				Out_uiAktSchritt := In_uiSchritt_09;
			ELSIF	(InOut_uiStatus_10 <> 0)
					AND (InOut_uiStatus_10 <> 4) THEN
				Out_uiAktSchritt := In_uiSchritt_10;				
			ELSIF	(InOut_uiStatus_11 <> 0)						(* 2014-07 gt: RDK90 *)
					AND (InOut_uiStatus_11 <> 4) THEN				(* 2014-07 gt: RDK90 *)
				Out_uiAktSchritt := In_uiSchritt_11;				(* 2014-07 gt: RDK90 *)
			ELSIF	(InOut_uiStatus_12 <> 0)						(* 2014-07 gt: RDK90 *)
					AND (InOut_uiStatus_12 <> 4) THEN				(* 2014-07 gt: RDK90 *)
				Out_uiAktSchritt := In_uiSchritt_12;				(* 2014-07 gt: RDK90 *)
			ELSIF	(InOut_uiStatus_13 <> 0)						(* 2014-07 gt: RDK90 *)
					AND (InOut_uiStatus_13 <> 4) THEN				(* 2014-07 gt: RDK90 *)
				Out_uiAktSchritt := In_uiSchritt_13;				(* 2014-07 gt: RDK90 *)
			ELSIF	(InOut_uiStatus_14 <> 0)						(* 2014-07 gt: RDK90 *)
					AND (InOut_uiStatus_14 <> 4) THEN				(* 2014-07 gt: RDK90 *)
				Out_uiAktSchritt := In_uiSchritt_14;				(* 2014-07 gt: RDK90 *)
			ELSIF	(InOut_uiStatus_15 <> 0)						(* 2014-07 gt: RDK90 *)
					AND (InOut_uiStatus_15 <> 4) THEN				(* 2014-07 gt: RDK90 *)
				Out_uiAktSchritt := In_uiSchritt_15;				(* 2014-07 gt: RDK90 *)
			ELSIF	(InOut_uiStatus_16 <> 0)						(* 2014-07 gt: RDK90 *)
					AND (InOut_uiStatus_16 <> 4) THEN				(* 2014-07 gt: RDK90 *)
				Out_uiAktSchritt := In_uiSchritt_16;				(* 2014-07 gt: RDK90 *)
			ELSIF	(InOut_uiStatus_17 <> 0)						(* 2014-07 gt: RDK90 *)
					AND (InOut_uiStatus_17 <> 4) THEN				(* 2014-07 gt: RDK90 *)
				Out_uiAktSchritt := In_uiSchritt_17;				(* 2014-07 gt: RDK90 *)
			ELSIF	(InOut_uiStatus_18 <> 0)						(* 2016-09 gt: *)
					AND (InOut_uiStatus_18 <> 4) THEN				(* 2016-09 gt: *)
				Out_uiAktSchritt := In_uiSchritt_18;				(* 2016-09 gt: *)
			ELSIF	(uiStatus_19_in_out <> 0)						(* 2016-09 gt: *)
					AND (uiStatus_19_in_out <> 4) THEN				(* 2016-09 gt: *)
				Out_uiAktSchritt := In_uiSchritt_19;				(* 2016-09 gt: *)
			ELSIF	(uiStatus_20_in_out <> 0)						(* 2016-09 gt: *)
					AND (uiStatus_20_in_out <> 4) THEN				(* 2016-09 gt: *)
				Out_uiAktSchritt := In_uiSchritt_20;				(* 2016-09 gt: *)
			ELSIF	(uiStatus_21_in_out <> 0)						(* 2016-09 gt: *)
					AND (uiStatus_21_in_out <> 4) THEN				(* 2016-09 gt: *)
				Out_uiAktSchritt := In_uiSchritt_21;				(* 2016-09 gt: *)
			END_IF
	ELSE Out_uiAktSchritt := 0;								
	END_IF
	(********************************************************************************************************************************************************)
	(* Transition / Weiterschaltung, wenn Einzelschritte beendet oder nicht relevant ************************************************************************)
	IF	TRUE
		AND	(	InOut_uiStatus_01 = 0
				OR InOut_uiStatus_01 = 3
				OR InOut_uiStatus_01 = 4								(* input/output: Status "1" *)
			)
		AND	(	InOut_uiStatus_02 = 0
				OR InOut_uiStatus_02 = 3
				OR InOut_uiStatus_02 = 4								(* input/output: Status "1" *)
			)		
		AND	(	InOut_uiStatus_03 = 0
				OR InOut_uiStatus_03 = 3
				OR InOut_uiStatus_03 = 4								(* input/output: Status "1" *)
			)
		AND	(	InOut_uiStatus_04 = 0
				OR InOut_uiStatus_04 = 3
				OR InOut_uiStatus_04 = 4								(* input/output: Status "1" *)
			)		
		AND	(	InOut_uiStatus_05 = 0
				OR InOut_uiStatus_05 = 3
				OR InOut_uiStatus_05 = 4								(* input/output: Status "1" *)
			)		
		AND	(	InOut_uiStatus_06 = 0
				OR InOut_uiStatus_06 = 3
				OR InOut_uiStatus_06 = 4								(* input/output: Status "1" *)
			)		
		AND	(	InOut_uiStatus_07 = 0
				OR InOut_uiStatus_07 = 3
				OR InOut_uiStatus_07 = 4								(* input/output: Status "1" *)
			)		
		AND	(	uiStatus_08_in_out = 0
				OR uiStatus_08_in_out = 3
				OR uiStatus_08_in_out = 4								(* input/output: Status "1" *)
			)		
		AND	(	InOut_uiStatus_09 = 0
				OR InOut_uiStatus_09 = 3
				OR InOut_uiStatus_09 = 4								(* input/output: Status "1" *)
			)		
		AND	(	InOut_uiStatus_10 = 0
				OR InOut_uiStatus_10 = 3
				OR InOut_uiStatus_10 = 4								(* input/output: Status "1" *)
			)
		AND	(	InOut_uiStatus_11 = 0																		(* 2014-07 gt: RDK90 *)
				OR InOut_uiStatus_11 = 3																	(* 2014-07 gt: RDK90 *)
				OR InOut_uiStatus_11 = 4								(* input/output: Status "1" *)		(* 2014-07 gt: RDK90 *)
			)																
		AND	(	InOut_uiStatus_12 = 0																		(* 2014-07 gt: RDK90 *)
				OR InOut_uiStatus_12 = 3																	(* 2014-07 gt: RDK90 *)
				OR InOut_uiStatus_12 = 4								(* input/output: Status "1" *)		(* 2014-07 gt: RDK90 *)
			)	
		AND	(	InOut_uiStatus_13 = 0																		(* 2014-07 gt: RDK90 *)
				OR InOut_uiStatus_13 = 3																	(* 2014-07 gt: RDK90 *)
				OR InOut_uiStatus_13 = 4								(* input/output: Status "1" *)		(* 2014-07 gt: RDK90 *)
			)	
		AND	(	InOut_uiStatus_14 = 0																		(* 2014-07 gt: RDK90 *)
				OR InOut_uiStatus_14 = 3																	(* 2014-07 gt: RDK90 *)
				OR InOut_uiStatus_14 = 4								(* input/output: Status "1" *)		(* 2014-07 gt: RDK90 *)
			)	
		AND	(	InOut_uiStatus_15 = 0																		(* 2014-07 gt: RDK90 *)
				OR InOut_uiStatus_15 = 3																	(* 2014-07 gt: RDK90 *)
				OR InOut_uiStatus_15 = 4								(* input/output: Status "1" *)		(* 2014-07 gt: RDK90 *)
			)
		AND	(	InOut_uiStatus_16 = 0																		(* 2014-07 gt: RDK90 *)
				OR InOut_uiStatus_16 = 3																	(* 2014-07 gt: RDK90 *)
				OR InOut_uiStatus_16 = 4								(* input/output: Status "1" *)		(* 2014-07 gt: RDK90 *)
			)
		AND	(	InOut_uiStatus_17 = 0																		(* 2014-07 gt: RDK90 *)
				OR InOut_uiStatus_17 = 3																	(* 2014-07 gt: RDK90 *)
				OR InOut_uiStatus_17 = 4								(* input/output: Status "1" *)		(* 2014-07 gt: RDK90 *)
			)
		AND	(	InOut_uiStatus_18 = 0																		(* 2016-09 gt: *)
				OR InOut_uiStatus_18 = 3																	(* 2016-09 gt: *)
				OR InOut_uiStatus_18 = 4								(* input/output: Status "1" *)		(* 2016-09 gt: *)
			)
		AND	(	uiStatus_19_in_out = 0																		(* 2016-09 gt: *)
				OR uiStatus_19_in_out = 3																	(* 2016-09 gt: *)
				OR uiStatus_19_in_out = 4								(* input/output: Status "1" *)		(* 2016-09 gt: *)
			)
		AND	(	uiStatus_20_in_out = 0																		(* 2016-09 gt: *)
				OR uiStatus_20_in_out = 3																	(* 2016-09 gt: *)
				OR uiStatus_20_in_out = 4								(* input/output: Status "1" *)		(* 2016-09 gt: *)
			)
		AND	(	uiStatus_21_in_out = 0																		(* 2016-09 gt: *)
				OR uiStatus_21_in_out = 3																	(* 2016-09 gt: *)
				OR uiStatus_21_in_out = 4								(* input/output: Status "1" *)		(* 2016-09 gt: *)
			) THEN		
		Out_bTransistion := TRUE;		
		Out_uiAktSchritt := In_uiSchrittTransition;					(* Schrittnummer für die Transition nach Blockquittierung, wenn also der Block abgearbeitet ist *)
	ELSE
		Out_bTransistion := FALSE;
	END_IF
ELSE
	In_uiSchritt_01					:= 0;								(* input: Schrittnummer "1" *)
	In_uiSchritt_02					:= 0;								(* input: Schrittnummer "2" *)
	In_uiSchritt_03					:= 0;								(* input: Schrittnummer "3" *)
	In_uiSchritt_04					:= 0;								(* input: Schrittnummer "4" *)
	In_uiSchritt_05					:= 0;								(* input: Schrittnummer "5" *)
	In_uiSchritt_06					:= 0;								(* input: Schrittnummer "6" *)	
	In_uiSchritt_07					:= 0;								(* input: Schrittnummer "7" *)
	In_uiSchritt_08					:= 0;								(* input: Schrittnummer "8" *)
	In_uiSchritt_09					:= 0;								(* input: Schrittnummer "9" *)
	In_uiSchritt_10					:= 0;								(* input: Schrittnummer "10" *)	
	In_uiSchritt_11					:= 0;								(* input: Schrittnummer "11" *)			(* 2014-07 gt: RDK90 *)
	In_uiSchritt_12					:= 0;								(* input: Schrittnummer "12" *)			(* 2014-07 gt: RDK90 *)
	In_uiSchritt_13					:= 0;								(* input: Schrittnummer "13" *)			(* 2014-07 gt: RDK90 *)
	In_uiSchritt_14					:= 0;								(* input: Schrittnummer "14" *)			(* 2014-07 gt: RDK90 *)
	In_uiSchritt_15					:= 0;								(* input: Schrittnummer "15" *)			(* 2014-07 gt: RDK90 *)
	In_uiSchritt_16					:= 0;								(* input: Schrittnummer "16" *)			(* 2014-07 gt: RDK90 *)
	In_uiSchritt_17					:= 0;								(* input: Schrittnummer "17" *)			(* 2014-07 gt: RDK90 *)
	In_uiSchritt_18					:= 0;								(* input: Schrittnummer "18" *)			(* 2016-09 gt: *)
	In_uiSchritt_19					:= 0;								(* input: Schrittnummer "19" *)			(* 2016-09 gt: *)
	In_uiSchritt_20					:= 0;								(* input: Schrittnummer "20" *)			(* 2016-09 gt: *)
	In_uiSchritt_21					:= 0;								(* input: Schrittnummer "21" *)			(* 2016-09 gt: *)	

	InOut_bQuit_01					:= FALSE;							(* input/output: Quittierung "1" *)
	InOut_uiStatus_01				:= 0;								(* input/output: Status "1" *)
	InOut_bQuit_02					:= FALSE;							(* input/output: Quittierung "2" *)	
	InOut_uiStatus_02				:= 0;								(* input/output: Status "2" *)
	InOut_bQuit_03					:= FALSE;							(* input/output: Quittierung "3" *)
	InOut_uiStatus_03				:= 0;								(* input/output: Status "3" *)
	InOut_bQuit_04					:= FALSE;							(* input/output: Quittierung "4" *)	
	InOut_uiStatus_04				:= 0;								(* input/output: Status "4" *)
	InOut_bQuit_05					:= FALSE;							(* input/output: Quittierung "5" *)
	InOut_uiStatus_05				:= 0;								(* input/output: Status "5" *)
	InOut_bQuit_06					:= FALSE;							(* input/output: Quittierung "6" *)	
	InOut_uiStatus_06				:= 0;								(* input/output: Status "6" *)
	InOut_bQuit_07					:= FALSE;							(* input/output: Quittierung "7" *)
	InOut_uiStatus_07				:= 0;								(* input/output: Status "7" *)
	InOut_bQuit_08					:= FALSE;							(* input/output: Quittierung "8" *)	
	uiStatus_08_in_out				:= 0;								(* input/output: Status "8" *)
	InOut_bQuit_09					:= FALSE;							(* input/output: Quittierung "9" *)
	InOut_uiStatus_09				:= 0;								(* input/output: Status "9" *)
	InOut_bQuit_10					:= FALSE;							(* input/output: Quittierung "10" *)		
	InOut_uiStatus_10				:= 0;								(* input/output: Status "10" *)
	InOut_bQuit_11					:= FALSE;							(* input/output: Quittierung "11" *)	(* 2014-07 gt: RDK90 *)		
	InOut_uiStatus_11				:= 0;								(* input/output: Status "11" *)			(* 2014-07 gt: RDK90 *)
	InOut_bQuit_12					:= FALSE;							(* input/output: Quittierung "12" *)	(* 2014-07 gt: RDK90 *)	
	InOut_uiStatus_12				:= 0;								(* input/output: Status "12" *)			(* 2014-07 gt: RDK90 *)
	InOut_bQuit_13					:= FALSE;							(* input/output: Quittierung "13" *)	(* 2014-07 gt: RDK90 *)	
	InOut_uiStatus_13				:= 0;								(* input/output: Status "13" *)			(* 2014-07 gt: RDK90 *)
	InOut_bQuit_14					:= FALSE;							(* input/output: Quittierung "14" *)	(* 2014-07 gt: RDK90 *)	
	InOut_uiStatus_14				:= 0;								(* input/output: Status "14" *)			(* 2014-07 gt: RDK90 *)
	InOut_bQuit_15					:= FALSE;							(* input/output: Quittierung "15" *)	(* 2014-07 gt: RDK90 *)	
	InOut_uiStatus_15				:= 0;								(* input/output: Status "15" *)			(* 2014-07 gt: RDK90 *)
	InOut_bQuit_16					:= FALSE;							(* input/output: Quittierung "16" *)	(* 2014-07 gt: RDK90 *)	
	InOut_uiStatus_16				:= 0;								(* input/output: Status "16" *)			(* 2014-07 gt: RDK90 *)	
	InOut_bQuit_17					:= FALSE;							(* input/output: Quittierung "17" *)	(* 2014-07 gt: RDK90 *)	
	InOut_uiStatus_17				:= 0;								(* input/output: Status "17" *)			(* 2014-07 gt: RDK90 *)
	InOut_bQuit_18					:= FALSE;							(* input/output: Quittierung "18" *)	(* 2016-09 gt: *)	
	InOut_uiStatus_18				:= 0;								(* input/output: Status "18" *)			(* 2016-09 gt: *)
	bQuit_19_in_out					:= FALSE;							(* input/output: Quittierung "19" *)	(* 2016-09 gt: *)	
	uiStatus_19_in_out				:= 0;								(* input/output: Status "19" *)			(* 2016-09 gt: *)
	bQuit_20_in_out					:= FALSE;							(* input/output: Quittierung "20" *)	(* 2016-09 gt: *)	
	uiStatus_20_in_out				:= 0;								(* input/output: Status "20" *)			(* 2016-09 gt: *)
	bQuit_21_in_out					:= FALSE;							(* input/output: Quittierung "21" *)	(* 2016-09 gt: *)	
	uiStatus_21_in_out				:= 0;								(* input/output: Status "21" *)			(* 2016-09 gt: *)	
	
	Out_uiAktSchritt				:= 0;								(* output: Aktueller Schritt aufgrund der "höchswertigsten" Quittierung  *)
	Out_bTransistion				:= FALSE;							(* output: Transition / Weiterschaltung, wenn Einzelschritte beendet oder nicht relevant *)	
END_IF	
(********************************************************************************************************************************************************)

END_FUNCTION_BLOCK

// GeneralFunctionBlocks/FB_ClockMarker
{attribute 'qualified_only' := ''}
{attribute 'namespace' := 'ILGStdLib.FunctionBlocks'}
FUNCTION_BLOCK FB_ClockMarker
VAR_OUTPUT
	/// Ausgangsvariable, die in der anparametrierten rRDM_Taktzeit_gb taktet 
	Out_bClock: BOOL;
	/// Ausgangsvariable, die in der anparametrierten rRDM_Taktzeit_gb einen Impuls abgibt 
	Out_bPulse: BOOL;
END_VAR
VAR
	/// Funktionsbaustein "Einschaltverzoegerung" fuer den Taktmerker 
	fbTonClock1: TON;
	/// Funktionsbaustein "Einschaltverzoegerung" fuer den Taktmerker 
	fbTonClock2: TON;
	/// Funktionsbaustein positive Flanke für Taktmerker 
	rtrig_Clock: R_TRIG;
END_VAR
VAR_INPUT
	/// Ansteuersignal fuer den Start des Funktionsbausteins / das Erzeugen das Taktimpulses 
	In_bEnable: BOOL;
	/// Anzuparametrierende Zeit, fuer die rRDM_Taktzeit_gb 
	In_tCycleTime: TIME;
END_VAR

(* #################################################################################################################### *)
(* ##   iLLiG_FB_Taktmerker	    																				 	 ## *)
(* ##																												 ## *)
(* ##	Dieser Funktionsbaustein erzeugt ein taktendes Ausgangssignal, in Abhaengigkeit der anparametrierten	     ## *)
(* ##	Zeitdauer.																									 ## *)
(* ##																												 ## *)
(* ##   Versions-History:																							 ## *)
(* ##   06. Dezember 2011		Version 1.0		-	erste Version.													 ## *)
(* ##																												 ## *)
(* ##																												 ## *)
(* #################################################################################################################### *)


(* -------------------------------------------------------------------------------------------------------------------- *)
(* -- Erzeugen des Taktsignals ---------------------------------------------------------------------------------------- *)	
(* -------------------------------------------------------------------------------------------------------------------- *)

IF In_bEnable THEN

	fbTonClock1(IN:= (NOT Out_bClock), PT:= In_tCycleTime, Q=> , ET=> );					(* Aufruf der Einschaltverzoegerung 1 *)
		
	fbTonClock2(IN:= (Out_bClock), PT:= In_tCycleTime, Q=> , ET=> );						(* Aufruf der Einschaltverzoegerung 2 *)
	
	IF fbTonClock1.Q THEN
		Out_bClock := TRUE;																(* Ausgang setzen *)
	ELSIF fbTonClock2.Q THEN
		Out_bClock := FALSE;																(* Ausgang zurueck setzen *)
	END_IF
	
	(* Impuls von Takt bilden *)
	rtrig_Clock(CLK:= Out_bClock);
	Out_bPulse := rtrig_Clock.Q;
	
ELSE
	Out_bClock		:= FALSE;															(* Ausgang abloeschen *)
	fbTonClock1(IN:= FALSE, PT:= In_tCycleTime, Q=> , ET=> );							(* Funktionsbaustein zurueck setzen *)
	fbTonClock2(IN:= FALSE, PT:= In_tCycleTime, Q=> , ET=> );							(* Funktionsbaustein zurueck setzen *)
END_IF

END_FUNCTION_BLOCK

// GeneralFunctionBlocks/FB_Convert8BitTo5BitParameter
{attribute 'qualified_only' := ''}
{attribute 'namespace' := 'ILGStdLib.FunctionBlocks'}
FUNCTION_BLOCK FB_Convert8BitTo5BitParameter
VAR_OUTPUT
	Out_dwOutput: DWORD;
	Out_bDone: BOOL;
	Out_bError: BOOL;
	Out_bActive: BOOL;
END_VAR
VAR
	udiTemp: UDINT;
	udiInput: UDINT;
	iStep: INT;
END_VAR
VAR_INPUT
	In_diInput: DINT;
	In_udiMask: UDINT;
	In_bEnable: BOOL;
	In_bStart: BOOL;
END_VAR

(* #################################################################################################################### *)
(* ##   iLLiG_FB_Bremspruefung    																				 	 ## *)
(* ##																											     ## *)
(* ##   erstellt von:																								 ## *)
(* ##   Markus Pfisterer, EE																						 ## *)
(* ##																											     ## *)
(* ##   Versions-History:																							 ## *)
(* ##   12.Oktober 2018		Version 1.0		-	Erste Version, nach Bereinigung der Fehler							 ## *)
(* #################################################################################################################### *)

(*
Funktionsbeschreibung:
Der Baustein konvertiert den Parameter S-0-0390 in ein bekanntes fünfstelliges Format.
*)


(* ####################################################################################################################################### *)
IF In_bEnable THEN
	(* #################################################### *)
	(* Start der Schritkette *)
	IF In_bStart AND NOT Out_bActive THEN
		iStep := 10;
	END_IF

	(* #################################################### *)
	(* Statusmeldung bilden *)
	IF iStep > 0 THEN
		Out_bActive := TRUE;
	ELSE
		Out_bActive := FALSE;
	END_IF


	(* #################################################### *)
	(* Schrittkette zur Konvertierung *)
	CASE iStep OF
	
		(* Initialisierung des Bausteins *)
		10:
			Out_bDone  := FALSE;
			Out_bError := FALSE;
			iStep 	 := 20;
			
		(* Konvertierung *)
		20:
			udiInput := DINT_TO_UDINT(In_diInput AND 16#000FFFFF);
			
			IF udiInput > 16#000F0000 THEN					// Error
				udiTemp := udiInput AND 16#00FF0000;			// Check if Error comes from IndraDrive 
				IF udiTemp = 16#F0000 THEN
					udiInput := udiInput AND In_udiMask;
					Out_dwOutput := udiInput + 16#000F0000;
					Out_bDone    := TRUE;
				ELSE
					Out_dwOutput := DINT_TO_DWORD(16#0);
					Out_bError    := TRUE;	
				END_IF	
				
			ELSIF udiInput > 16#000E0000 THEN				// Warning
				udiTemp := udiInput AND  16#00FF0000;			// Check if Error comes from IndraDrive 
				IF udiTemp = 16#E0000 THEN
					udiInput := udiInput AND In_udiMask;
					Out_dwOutput := udiInput + 16#000E0000;
					Out_bDone    := TRUE;
				ELSE
					Out_dwOutput := DINT_TO_DWORD(16#0);	
					Out_bError    := TRUE;	
				END_IF	
			ELSIF udiInput > 16#000C0000 THEN				// Diagnosis
				udiTemp := udiInput AND  16#00FF0000;			// Check if Error comes from IndraDrive 
				IF udiTemp = 16#C0000 THEN
					udiInput := udiInput AND In_udiMask;
					Out_dwOutput := udiInput + 16#000C0000;
					Out_bDone    := TRUE;
				ELSE
					Out_dwOutput := DINT_TO_DWORD(16#0);
					Out_bError    := TRUE;		
				END_IF
			ELSIF udiInput > 16#000A0000 THEN				// Status
				udiTemp := udiInput AND  16#00FF0000;			// Check if Error comes from IndraDrive 
				IF udiTemp = 16#A0000 THEN
					udiInput := udiInput AND In_udiMask;
					Out_dwOutput := udiInput + 16#000A0000;
					Out_bDone    := TRUE;
				ELSE
					Out_dwOutput := DINT_TO_DWORD(16#0);
					Out_bError    := TRUE;		
				END_IF
				
			ELSE
				Out_bError := TRUE;	
			END_IF
	
			Out_bActive := FALSE;
			iStep 	  := 0;
	END_CASE
END_IF

END_FUNCTION_BLOCK

// GeneralFunctionBlocks/FB_IlligOperatingModes
{attribute 'qualified_only' := ''}
{attribute 'namespace' := 'ILGStdLib.FunctionBlocks'}
FUNCTION_BLOCK FB_IlligOperatingModes
VAR_OUTPUT
	/// Dummyvariable, da bei erster Variable keine Quick Info möglich 
	OUT_bDummy: BOOL;
	/// Betriebsart: "Referenzieren" (M12.7) 
	OUT_bBetriebsart_Ctrl_REFERENZIEREN: BOOL;
	/// Betriebsart: Vorwahl "Referenzieren" (M12.6) 
	OUT_bBetriebsart_Vorwahl_REFERENZIEREN: BOOL;
	/// Betriebsart: "Hand" (M13.0)
	OUT_bBetriebsart_Ctrl_HAND: BOOL;
	/// Betriebsart: "Ruesten" (M12.0) 
	OUT_bBetriebsart_Ctrl_RUESTEN: BOOL;
	/// Betriebsart: "Einruesten" (M12.1) 
	OUT_bBetriebsart_Ctrl_EINRUESTEN: BOOL;
	/// Betriebsart: "Ausruesten" (M12.2) 
	OUT_bBetriebsart_Ctrl_AUSRUESTEN: BOOL;
	/// Betriebsart: "VorwahlAuto" (M14.7)
	OUT_bBetriebsart_Ctrl_VORWAHLAUTO: BOOL;
	/// Betriebsart: "Automatik" oder "Startautomatik" ("M14.5" oder "M18.3")
	OUT_bBetriebsart_Ctrl_AUTOLAEUFT: BOOL;
	/// Betriebsart: "Automatik" (M14.0)
	OUT_bBetriebsart_Ctrl_AUTOMATIK: BOOL;
	/// Betriebsart: "Grundstellungsfahrt" (M14.4)
	OUT_bBetriebsart_Ctrl_GRUNDSTELLUNGSFAHRT: BOOL;
	/// Betriebsart: "Automatik Laeuft" und "Startautomatik" beendet (M14.5) 
	OUT_bBetriebsart_Ctrl_AUTOLAEUFT_STARTAUTO_fertig: BOOL;
	/// Betriebsart: "Schluesselschalter" (M11.7) 
	OUT_bBetriebsart_Ctrl_SCHLUESSELSCHALTER: BOOL;
	/// Betriebsart: Impuls Drucktaster "Start" (M11.0) 
	OUT_bImp_DT_Automatik_Start: BOOL;
	/// Betriebsart: Impuls "Automatik EIN" (M16.0) 
	OUT_bImp_Betriebsart_Ctrl_AUTOMATIK_EIN: BOOL;
	/// Betriebsart: Impuls "Automatik AUS" (M16.2) 
	OUT_bImp_Betriebsart_Ctrl_AUTOMATIK_AUS: BOOL;
	/// Betriebsart: Impuls "Automatik Laeuft" und "Startautomatik" beendet (M16.4) 
	OUT_bImp_Betriebsart_Ctrl_AUTOLAEUFT_STARTAUTO_fertig: BOOL;
	/// Betriebsart: "Automatik Aus" (nicht M14.0 und nicht M14.5) verzögert 1 Sek. 
	OUT_bBetriebsart_Automatik_Aus_Verz: BOOL;
	/// Betriebsart: Freigabe Hand (M13.1) 
	OUT_bFreig_Betriebsart_Hand: BOOL;
	/// Anforderung Stop in Grundstellung gespeichert 
	OUT_bAnf_StopGrdst_gesp: BOOL;
	/// Anzeige Betriebsart: 0= Hand, 1= Rüsten, 2= Einrüsten, 4= Ausrüsten, 8= Vorwahl Automatik, 16= Vorwahl Referenzieren 
	OUT_byAnzeige_Betriebsart: BYTE;
END_VAR
VAR
	/// Dummyvariable, da bei erster Variable keine Quick Info möglich 
	bDummy: BOOL;
	/// Bedienfeld Anwahl "Vorwahl Automatik" 
	bBBF_Anw_Betriebsart_Automatik: BOOL;
	/// Bedienfeld Anwahl Betriebsart Hand 
	bBBF_Anw_Betriebsart_Hand: BOOL;
	/// Impuls Grundstellungsfahrt beendet (M17.2) 
	bImpuls_GrdstFahrt_Beendet: BOOL;
	/// Freigabe Grundstellungsfahrt 
	bFreig_Grundstellungsfahrt: BOOL;
	/// Start Grundstellungsfahrt exter gespeichert 
	bStart_Grundstellungsfahrt_extern_gesp: BOOL;
	/// Anforderung Stop in Grundstellung gespeichert 
	bAnf_StopGrdst_gesp: BOOL;
	/// Dummyvariable, da bei erster Variable keine Quick Info möglich 
	rtrigDummy: R_TRIG;
	/// Positive Flanke Bedienfeld Anwahl Schlüsselschalter ( M19.6) 
	rtrigBetriebsart_Ctrl_Schluesselschalter: R_TRIG;
	/// Negative Flanke Bedienfeld Anwahl Schlüsselschalter ( M19.2) 
	ftrigBetriebsart_Ctrl_Schluesselschalter: F_TRIG;
	/// Positive Flanke Drucktaster Automatik Start (M11.0)
	rtrigDT_Automatik_Start: R_TRIG;
	/// Positive Flanke Drucktaster Automatik Stop (M11.2)
	rtrigDT_Automatik_Stop: R_TRIG;
	/// Positive Flanke Bedienfeld Anwahl Betriebsart Ruesten ( M27.0) 
	rtrigBBF_Anw_Betriebsart_Ruesten: R_TRIG;
	/// Positive Flanke Bedienfeld Anwahl Betriebsart Einruesten ( M27.1) 
	rtrigBBF_Anw_Betriebsart_Einruesten: R_TRIG;
	/// Positive Flanke Bedienfeld Anwahl Betriebsart Ausruesten ( M27.2) 
	rtrigBBF_Anw_Betriebsart_Ausruesten: R_TRIG;
	/// Positive Flanke Bedienfeld Anwahl Betriebsart Referenzieren ( M27.3) 
	rtrigBBF_Anw_Betriebsart_Referenzieren: R_TRIG;
	/// Hilfsmerker für Impuls Grundstellungsfahrt beendet 
	rtrigHM_Impuls_Grundstellungsfahrt_beendet: R_TRIG;
	/// Hilfsmerker Positive Flanke "Automatik EIN" 
	rtrigHM_Automatik_EIN: R_TRIG;
	/// Hilfsmerker Positive Flanke "Automatik AUS" 
	rtrigHM_Automatik_AUS: R_TRIG;
	/// Hilfsmerker Positive Flanke "Automatik läuft" 
	rtrigHM_Automatik_laeuft: R_TRIG;
	/// Hilfsmerker "Automatik AUS" verzögert 
	tonHM_Automatik_Aus: TON;
	/// Hilfsmerker Positive Flanke Impuls "Automatik Laeuft" und "Startautomatik" beendet 
	rtrigHM_AUTOLAEUFT_STARTAUTO_fertig: R_TRIG;
END_VAR
VAR_INPUT
	/// Dummyvariable, da bei erster Variable keine Quick Info möglich 
	IN_bDummy: BOOL;
	/// Drucktaster "Betriebsart Start" 
	IN_bDT_Betriebsart_Start: BOOL;
	/// Drucktaster "Betriebsart Stop" 
	IN_bDT_Betriebsart_Stop: BOOL;
	/// Schlüsselschalter 
	IN_bSCHLUESSELSCHALTER: BOOL;
	/// Bedienfeld Anwahl Betriebsart Ruesten ( M27.0) 
	IN_bBBF_Anw_Betriebsart_Ruesten: BOOL;
	/// Bedienfeld Anwahl Betriebsart Einruesten ( M27.1) 
	IN_bBBF_Anw_Betriebsart_Einruesten: BOOL;
	/// Bedienfeld Anwahl Betriebsart Ausruesten ( M27.2) 
	IN_bBBF_Anw_Betriebsart_Ausruesten: BOOL;
	/// Bedienfeld Anwahl Betriebsart Referenzieren ( M27.3) 
	IN_bBBF_Anw_Betriebsart_Referenzieren: BOOL;
	/// Linie in Grundstellung (RDM & Stapelung (M14.6) 
	IN_bLinie_In_Grundstellung: BOOL;
	/// Anforderung Vorwahl Automatik extern. Z.B. von Bremsprüfung 
	IN_bAnf_Vorwahl_Automatik_extern: BOOL;
	/// Schrittkette Werkzeugeinbau aktiv (M518.4) 
	IN_bSKWerkzeugeinbau_aktiv: BOOL;
	/// Schrittkette Werkzeugausbau aktiv (M537.7) 
	IN_bSKWerkzeugausbau_aktiv: BOOL;
	/// Ein- und Ausrüsten zurücksetzen 
	IN_bReset_Ein_Ausruesten_extern: BOOL;
	/// Anforderung Betriebsart Hand von extern z.B. von Bremsprüfung 
	IN_bAnf_Betriebsart_Hand_extern: BOOL;
	/// Reset Betriebsart Hand von extern z.B. von Bremsprüfung 
	IN_bReset_Betriebsart_Hand_extern: BOOL;
	/// Reset Vorwahl Automatik von extern z.B. von Bremsprüfung 
	IN_bReset_Vorwahl_Automatik_extern: BOOL;
	/// Freigabe Vorwahl Automatik 
	IN_bFreig_Vorwahl_Automatik_extern: BOOL;
	/// Stopp in Grundstellung Fehler aktiv 
	IN_bStopInGrundstellung: BOOL;
	/// Sofortstopfehler aktiv 
	IN_bSofortstopp: BOOL;
	/// Abläufe in Vorwahl Automatik aktiv z.B. Räumen 
	IN_bAblaeufe_Vorwahl_Automatik_aktiv: BOOL;
	/// Steuerstrom EIN (M10.0) 
	IN_bSteuerstrom_Ein: BOOL;
	/// Freigabe Grundstellungsfahrt 
	IN_bFreig_Grundstellungsfahrt_extern: BOOL;
	/// Freigabe Grundstellungsfahrt ohne Schlüsselschalter (Bsp. innerhalb des Rüstablaufs 
	IN_bFreig_GrdstFahrt_mit_SCHLUESSELSCHALTER_extern: BOOL;
	/// Grundstellungsfahrt löschen extern
	IN_bGrdstFahrt_loeschen_extern: BOOL;
	/// Anforderung Grundstellungsfahrt von Extern z.B.Bremsprüfung 
	IN_bAnf_Grundstellungsfahrt_Extern: BOOL;
	/// Reset Automatik von Extern z.B. Bremsprüfung, Schmierhub... 
	IN_bReset_Automatik_extern: BOOL;
	/// Freigabe Automatik 
	IN_bFreig_Automatik_extern: BOOL;
	/// Automatikabläufe der Linie nicht aktiv, Automatik läuft kann zurückgenommen werden 
	IN_bAutomatikablaeufe_nicht_Aktiv: BOOL;
	/// Freigabe "Automatik läuft" extern 
	IN_bFreig_Automatik_Laeuft_extern: BOOL;
	/// Freigabe "Automatik Stopp in Grundstellung" extern 
	IN_bFreig_Automatik_Stop_Grdst_extern: BOOL;
	/// Start "Automatik läuft" Extern 
	IN_bStart_Automatik_Laeuft_Extern: BOOL;
	/// Startautomatik läuft 
	IN_bStartautomatik_Laeuft: BOOL;
END_VAR


(*##########################################################################################################################################################################################################*)
(* Drucktaster, Schlüsselschalter, BBF-Anwahlen *)
(*##########################################################################################################################################################################################################*)

(* Positive Flanke Drucktaster "Start" *)
rtrigDT_Automatik_Start(CLK:= IN_bDT_Betriebsart_Start);

(* Positive Flanke Drucktaster "Stop" *)
rtrigDT_Automatik_Stop(CLK:= IN_bDT_Betriebsart_Stop);

(* Schluesselschalter eingeschaltet *)
OUT_bBetriebsart_Ctrl_SCHLUESSELSCHALTER := IN_bSCHLUESSELSCHALTER AND NOT OUT_bBetriebsart_Ctrl_AUTOLAEUFT;

(* Positive Flanke Bedienfeld Anwahl Schluesselschalter *)
rtrigBetriebsart_Ctrl_Schluesselschalter(CLK:= IN_bSCHLUESSELSCHALTER);

(* Negative Flanke Bedienfeld Anwahl Schluesselschalter *)
ftrigBetriebsart_Ctrl_Schluesselschalter(CLK:= IN_bSCHLUESSELSCHALTER);

(* Positive Flanke Bedienfeld Anwahl Betriebsart Ruesten *)
rtrigBBF_Anw_Betriebsart_Ruesten(CLK:= IN_bBBF_Anw_Betriebsart_Ruesten);

(* Positive Flanke Bedienfeld Anwahl Betriebsart Einruesten *)
rtrigBBF_Anw_Betriebsart_Einruesten(CLK:= IN_bBBF_Anw_Betriebsart_Einruesten);

(* Positive Flanke Bedienfeld Anwahl Betriebsart Ausruesten *)
rtrigBBF_Anw_Betriebsart_Ausruesten(CLK:= IN_bBBF_Anw_Betriebsart_Ausruesten);

(* Positive Flanke Bedienfeld Anwahl Betriebsart Referenzieren *)
rtrigBBF_Anw_Betriebsart_Referenzieren(CLK:= IN_bBBF_Anw_Betriebsart_Referenzieren);

(* Bedienfeld Anwahl Betriebsart Automatik *)
bBBF_Anw_Betriebsart_Automatik := IN_bLinie_In_Grundstellung AND	bImpuls_GrdstFahrt_Beendet AND IN_bFreig_Vorwahl_Automatik_extern;

(* Bedienfeld Anwahl Betriebsart Hand *)
bBBF_Anw_Betriebsart_Hand := NOT OUT_bBetriebsart_Ctrl_AUTOMATIK AND NOT OUT_bBetriebsart_Ctrl_GRUNDSTELLUNGSFAHRT AND NOT 
																OUT_bBetriebsart_Ctrl_AUTOLAEUFT AND NOT OUT_bBetriebsart_Ctrl_VORWAHLAUTO AND NOT
																OUT_bBetriebsart_Ctrl_SCHLUESSELSCHALTER AND NOT bBBF_Anw_Betriebsart_Automatik AND NOT
																IN_bAnf_Vorwahl_Automatik_extern;

(* Automatik Stopp speichern, um an einer definierten Stelle Stopp in Grundstellung einzuleiten *)
IF ((IN_bStopInGrundstellung OR IN_bReset_Automatik_extern OR rtrigDT_Automatik_Stop.Q) AND NOT IN_bFreig_Automatik_Stop_Grdst_extern) THEN
	bAnf_StopGrdst_gesp := TRUE;
END_IF
(* Sobald die Automatik aus ist, speicher wieder rücksetzen *)
IF NOT OUT_bBetriebsart_Ctrl_AUTOMATIK THEN
	bAnf_StopGrdst_gesp := FALSE;
END_IF																
(*##########################################################################################################################################################################################################*)
(* Betriebsarten *)
(*##########################################################################################################################################################################################################*)
(* ********************************************************************************************************************** *)
(* Ruesten *)
(* ********************************************************************************************************************** *)
(* Betriebsart: "Ruesten" *)
IF ((NOT OUT_bBetriebsart_Ctrl_SCHLUESSELSCHALTER) OR rtrigBBF_Anw_Betriebsart_Einruesten.Q OR rtrigBBF_Anw_Betriebsart_Ausruesten.Q OR
	rtrigBBF_Anw_Betriebsart_Referenzieren.Q) THEN

	OUT_bBetriebsart_Ctrl_RUESTEN:= FALSE;

ELSIF ((rtrigBBF_Anw_Betriebsart_Ruesten.Q AND NOT IN_bSKWerkzeugeinbau_aktiv AND NOT IN_bSKWerkzeugausbau_aktiv) OR
		rtrigBetriebsart_Ctrl_Schluesselschalter.Q OR (rtrigDT_Automatik_Stop.Q AND (OUT_bBetriebsart_Vorwahl_REFERENZIEREN OR
		OUT_bBetriebsart_Ctrl_REFERENZIEREN))) THEN 
		
	OUT_bBetriebsart_Ctrl_RUESTEN:= TRUE;
END_IF
(* ---------------------------------------------------------------------------------------------------------------------- *)
(* Betriebsart: "Einruesten" *)
IF ((NOT OUT_bBetriebsart_Ctrl_SCHLUESSELSCHALTER) OR ((rtrigBBF_Anw_Betriebsart_Ruesten.Q OR rtrigBBF_Anw_Betriebsart_Ausruesten.Q OR 
	rtrigBBF_Anw_Betriebsart_Referenzieren.Q) AND NOT IN_bSKWerkzeugeinbau_aktiv) OR IN_bReset_Ein_Ausruesten_extern) THEN

	OUT_bBetriebsart_Ctrl_EINRUESTEN:= FALSE;

ELSIF (rtrigBBF_Anw_Betriebsart_Einruesten.Q) THEN 

	OUT_bBetriebsart_Ctrl_EINRUESTEN:= TRUE;

END_IF
(* ---------------------------------------------------------------------------------------------------------------------- *)
(* Betriebsart: "Ausruesten" *)
IF ((NOT OUT_bBetriebsart_Ctrl_SCHLUESSELSCHALTER) OR ((rtrigBBF_Anw_Betriebsart_Ruesten.Q OR rtrigBBF_Anw_Betriebsart_Einruesten.Q OR 
	rtrigBBF_Anw_Betriebsart_Referenzieren.Q) AND NOT IN_bSKWerkzeugausbau_aktiv) OR IN_bReset_Ein_Ausruesten_extern) THEN

	OUT_bBetriebsart_Ctrl_AUSRUESTEN:= FALSE;

ELSIF (rtrigBBF_Anw_Betriebsart_Ausruesten.Q) THEN 

	OUT_bBetriebsart_Ctrl_AUSRUESTEN:= TRUE;

END_IF
(* ********************************************************************************************************************** *)
(* Referenzieren *)
(* ********************************************************************************************************************** *)
(* Betriebsart: "Vorwahl Referenzieren" *)
IF ((NOT OUT_bBetriebsart_Ctrl_SCHLUESSELSCHALTER) OR rtrigBBF_Anw_Betriebsart_Ruesten.Q OR	rtrigBBF_Anw_Betriebsart_Einruesten.Q OR 
	rtrigBBF_Anw_Betriebsart_Ausruesten.Q OR rtrigDT_Automatik_Stop.Q) THEN
			
	OUT_bBetriebsart_Vorwahl_REFERENZIEREN:= FALSE;

ELSIF ((rtrigBBF_Anw_Betriebsart_Referenzieren.Q) AND NOT IN_bSKWerkzeugeinbau_aktiv AND NOT IN_bSKWerkzeugausbau_aktiv) THEN 

	OUT_bBetriebsart_Vorwahl_REFERENZIEREN:= TRUE;

END_IF
(* ---------------------------------------------------------------------------------------------------------------------- *)
(* Betriebsart: "Referenzieren" *)
IF ((NOT OUT_bBetriebsart_Ctrl_SCHLUESSELSCHALTER) OR NOT OUT_bBetriebsart_Vorwahl_REFERENZIEREN OR rtrigDT_Automatik_Stop.Q) THEN

	OUT_bBetriebsart_Ctrl_REFERENZIEREN:= FALSE;

ELSIF ((rtrigDT_Automatik_Start.Q) AND OUT_bBetriebsart_Vorwahl_REFERENZIEREN) THEN 

	OUT_bBetriebsart_Ctrl_REFERENZIEREN:= TRUE;

END_IF
(* ********************************************************************************************************************** *)
(* Hand *)
(* ********************************************************************************************************************** *)
(* Betriebsart: "Hand" *)
IF ((OUT_bBetriebsart_Ctrl_SCHLUESSELSCHALTER) OR IN_bReset_Betriebsart_Hand_extern OR OUT_bBetriebsart_Ctrl_GRUNDSTELLUNGSFAHRT OR
	bBBF_Anw_Betriebsart_Automatik) THEN
	
	OUT_bBetriebsart_Ctrl_HAND:= FALSE;

ELSIF (IN_bAnf_Betriebsart_Hand_extern OR bBBF_Anw_Betriebsart_Hand OR (ftrigBetriebsart_Ctrl_Schluesselschalter.Q)) THEN

	OUT_bBetriebsart_Ctrl_HAND:= TRUE;

END_IF
(* ********************************************************************************************************************** *)
(* Automatik *)
(* ********************************************************************************************************************** *)
(* Betriebsart: "Vorwahl Automatik" *)
IF (OUT_bBetriebsart_Ctrl_SCHLUESSELSCHALTER OR IN_bAnf_Betriebsart_Hand_extern OR bBBF_Anw_Betriebsart_Hand OR
	((rtrigDT_Automatik_Stop.Q OR (IN_bStopInGrundstellung AND IN_bLinie_In_Grundstellung AND NOT IN_bAblaeufe_Vorwahl_Automatik_aktiv) OR 
	OUT_bBetriebsart_Ctrl_GRUNDSTELLUNGSFAHRT OR 
	(NOT IN_bLinie_In_Grundstellung AND NOT IN_bAblaeufe_Vorwahl_Automatik_aktiv)) AND NOT OUT_bBetriebsart_Ctrl_AUTOMATIK AND
	 NOT OUT_bBetriebsart_Ctrl_AUTOLAEUFT)) THEN
	
	OUT_bBetriebsart_Ctrl_VORWAHLAUTO:= FALSE;

ELSIF ((IN_bAnf_Vorwahl_Automatik_extern OR bBBF_Anw_Betriebsart_Automatik) AND IN_bFreig_Vorwahl_Automatik_extern AND
	NOT IN_bStopInGrundstellung) THEN
	
	OUT_bBetriebsart_Ctrl_VORWAHLAUTO:= TRUE;

END_IF
(* ---------------------------------------------------------------------------------------------------------------------- *)
(* Impuls Grundstellungsfahrt beendet und Maschine in Grundstellung *)
rtrigHM_Impuls_Grundstellungsfahrt_beendet(CLK:=  (NOT (rtrigDT_Automatik_Start.Q) AND NOT OUT_bBetriebsart_Ctrl_GRUNDSTELLUNGSFAHRT));
bImpuls_GrdstFahrt_Beendet := (rtrigHM_Impuls_Grundstellungsfahrt_beendet.Q AND IN_bLinie_In_Grundstellung);
(* ---------------------------------------------------------------------------------------------------------------------- *)
(* Freigabe Grundstellungsfahrt *)
bFreig_Grundstellungsfahrt := IN_bFreig_Grundstellungsfahrt_extern AND NOT IN_bLinie_In_Grundstellung;
(* ---------------------------------------------------------------------------------------------------------------------- *)
(* Betriebsart: "Grundstellungsfahrt" *)
IF ((OUT_bBetriebsart_Ctrl_SCHLUESSELSCHALTER AND NOT IN_bFreig_GrdstFahrt_mit_SCHLUESSELSCHALTER_extern) OR IN_bStopInGrundstellung OR IN_bSofortstopp OR OUT_bBetriebsart_Ctrl_AUTOMATIK OR
	rtrigDT_Automatik_Stop.Q OR NOT IN_bSteuerstrom_Ein OR OUT_bBetriebsart_Ctrl_AUTOLAEUFT OR (IN_bGrdstFahrt_loeschen_extern AND bStart_Grundstellungsfahrt_extern_gesp)OR 
	(OUT_bBetriebsart_Ctrl_GRUNDSTELLUNGSFAHRT AND IN_bLinie_In_Grundstellung)) THEN

	OUT_bBetriebsart_Ctrl_GRUNDSTELLUNGSFAHRT:= FALSE;
	bStart_Grundstellungsfahrt_extern_gesp := FALSE;

ELSIF ((rtrigDT_Automatik_Start.Q OR IN_bAnf_Grundstellungsfahrt_Extern) AND bFreig_Grundstellungsfahrt) THEN
	
	(* Merken wenn Grundstellungsfahrt von extern angefordert wurde *)
	IF IN_bAnf_Grundstellungsfahrt_Extern THEN
		bStart_Grundstellungsfahrt_extern_gesp := TRUE;
	END_IF
	OUT_bBetriebsart_Ctrl_GRUNDSTELLUNGSFAHRT:= TRUE;

END_IF
(* ---------------------------------------------------------------------------------------------------------------------- *)
(* Betriebsart: "Automatik" *)
IF (((IN_bStopInGrundstellung OR IN_bReset_Automatik_extern OR rtrigDT_Automatik_Stop.Q OR bAnf_StopGrdst_gesp) AND IN_bFreig_Automatik_Stop_Grdst_extern) OR IN_bSofortstopp OR
	NOT IN_bSteuerstrom_Ein OR NOT OUT_bBetriebsart_Ctrl_VORWAHLAUTO OR OUT_bBetriebsart_Ctrl_GRUNDSTELLUNGSFAHRT OR
	OUT_bBetriebsart_Vorwahl_REFERENZIEREN) THEN
	
	OUT_bBetriebsart_Ctrl_AUTOMATIK:= FALSE;

ELSIF (rtrigDT_Automatik_Start.Q AND IN_bFreig_Automatik_extern AND IN_bLinie_In_Grundstellung) THEN

	OUT_bBetriebsart_Ctrl_AUTOMATIK:= TRUE;

END_IF
(* ---------------------------------------------------------------------------------------------------------------------- *)
(* Betriebsart: "Startautomatik laeuft" *)
IF (IN_bSofortstopp OR NOT IN_bSteuerstrom_Ein OR	NOT OUT_bBetriebsart_Ctrl_VORWAHLAUTO OR (NOT OUT_bBetriebsart_Ctrl_AUTOMATIK AND
	IN_bLinie_In_Grundstellung AND IN_bAutomatikablaeufe_nicht_Aktiv)) THEN
				
	OUT_bBetriebsart_Ctrl_AUTOLAEUFT_STARTAUTO_fertig:= FALSE;

ELSIF IN_bStart_Automatik_Laeuft_Extern AND IN_bFreig_Automatik_Laeuft_extern AND OUT_bBetriebsart_Ctrl_AUTOMATIK THEN
	
	OUT_bBetriebsart_Ctrl_AUTOLAEUFT_STARTAUTO_fertig:= TRUE;

END_IF
(* ---------------------------------------------------------------------------------------------------------------------- *)
(* Betriebsart: "Automatik läuft" (M14.5) oder (M18.3) *)
OUT_bBetriebsart_Ctrl_AUTOLAEUFT := OUT_bBetriebsart_Ctrl_AUTOLAEUFT_STARTAUTO_fertig OR IN_bStartautomatik_Laeuft;
(*##########################################################################################################################################################################################################*)
(* Zustaende *)
(*##########################################################################################################################################################################################################*)
(* Positive Flanke Drucktaster "Start" *)
OUT_bImp_DT_Automatik_Start := rtrigDT_Automatik_Start.Q;
(* Positive Flanke "Automatik Ein" (M16.0) *)
rtrigHM_Automatik_EIN(CLK:= OUT_bBetriebsart_Ctrl_AUTOMATIK);
OUT_bImp_Betriebsart_Ctrl_AUTOMATIK_EIN := rtrigHM_Automatik_EIN.Q;
(* ---------------------------------------------------------------------------------------------------------------------- *)
(* Positive Flanke "Automatik AUS" (M16.2) *)
rtrigHM_Automatik_AUS(CLK:= (NOT OUT_bBetriebsart_Ctrl_AUTOMATIK AND NOT OUT_bBetriebsart_Ctrl_AUTOLAEUFT_STARTAUTO_fertig AND 
															NOT OUT_bBetriebsart_Ctrl_VORWAHLAUTO));
OUT_bImp_Betriebsart_Ctrl_AUTOMATIK_AUS := rtrigHM_Automatik_AUS.Q;
(* ---------------------------------------------------------------------------------------------------------------------- *)
(* Positive Flanke "Automatik laeuft, Startautomatik beendet" (M16.4) *)
rtrigHM_AUTOLAEUFT_STARTAUTO_fertig(CLK:= OUT_bBetriebsart_Ctrl_AUTOLAEUFT_STARTAUTO_fertig);
OUT_bImp_Betriebsart_Ctrl_AUTOLAEUFT_STARTAUTO_fertig := rtrigHM_AUTOLAEUFT_STARTAUTO_fertig.Q;
(* ---------------------------------------------------------------------------------------------------------------------- *)
(* Betriebsart: "Automatik Aus" (nicht M14.0 und nicht M14.5) verzögert 400ms (M16.6) *)
(* 190903 Hauser: AND NOT bBetriebsart_Ctrl_AUTOLAEUFT_o hinzu, wenn touchen noch nicht erledigt sollen trotzdem die 400ms Verzögerung erst nach "Stopp in Grundstellung" ablaufen *)
tonHM_Automatik_Aus(IN:= (NOT OUT_bBetriebsart_Ctrl_AUTOMATIK AND NOT OUT_bBetriebsart_Ctrl_AUTOLAEUFT_STARTAUTO_fertig AND NOT OUT_bBetriebsart_Ctrl_AUTOLAEUFT), PT:=T#400MS, Q=> , ET=> );
OUT_bBetriebsart_Automatik_Aus_Verz := tonHM_Automatik_Aus.Q;
(* Anforderung Stopp in Grundstellung ist aktiv *)
OUT_bAnf_StopGrdst_gesp := bAnf_StopGrdst_gesp;
(* ---------------------------------------------------------------------------------------------------------------------- *)
(* Betriebsart: Freigabe Hand (M13.1) *)
OUT_bFreig_Betriebsart_Hand := NOT OUT_bBetriebsart_Ctrl_GRUNDSTELLUNGSFAHRT AND NOT OUT_bBetriebsart_Ctrl_VORWAHLAUTO AND
														 NOT OUT_bBetriebsart_Ctrl_AUTOMATIK AND NOT OUT_bBetriebsart_Ctrl_AUTOLAEUFT AND 
														 NOT IN_bSKWerkzeugeinbau_aktiv AND NOT IN_bSKWerkzeugausbau_aktiv;
(* ---------------------------------------------------------------------------------------------------------------------- *)
(* Betriebsart: Startautomatik aktiv (M18.3) *)
OUT_bFreig_Betriebsart_Hand := NOT OUT_bBetriebsart_Ctrl_GRUNDSTELLUNGSFAHRT AND NOT OUT_bBetriebsart_Ctrl_VORWAHLAUTO AND
														 NOT OUT_bBetriebsart_Ctrl_AUTOMATIK AND NOT OUT_bBetriebsart_Ctrl_AUTOLAEUFT AND 
														 NOT IN_bSKWerkzeugeinbau_aktiv AND NOT IN_bSKWerkzeugausbau_aktiv;
														 

(*##########################################################################################################################################################################################################*)
(* Visualisiserung *)
(*##########################################################################################################################################################################################################*)
(* Anzeige Betriebsart: 0= Hand, 1= Rüsten, 2= Einrüsten, 4= Ausrüsten, 8= Vorwahl Automatik, 16= Vorwahl Referenzieren *)
IF OUT_bBetriebsart_Ctrl_HAND THEN
	OUT_byAnzeige_Betriebsart := 0;
ELSIF OUT_bBetriebsart_Ctrl_RUESTEN THEN
	OUT_byAnzeige_Betriebsart := 1;
ELSIF OUT_bBetriebsart_Ctrl_EINRUESTEN AND NOT OUT_bBetriebsart_Ctrl_RUESTEN THEN
	OUT_byAnzeige_Betriebsart := 2;
ELSIF OUT_bBetriebsart_Ctrl_AUSRUESTEN AND NOT OUT_bBetriebsart_Ctrl_RUESTEN THEN
	OUT_byAnzeige_Betriebsart := 4;
ELSIF OUT_bBetriebsart_Ctrl_VORWAHLAUTO THEN
	OUT_byAnzeige_Betriebsart := 8;
ELSIF OUT_bBetriebsart_Vorwahl_REFERENZIEREN THEN
	OUT_byAnzeige_Betriebsart := 16;

END_IF

END_FUNCTION_BLOCK

// GeneralFunctionBlocks/FB_IlligZaehlstern
{attribute 'qualified_only' := ''}
{attribute 'namespace' := 'ILGStdLib.FunctionBlocks'}
FUNCTION_BLOCK FB_IlligZaehlstern
VAR_OUTPUT
	/// Fehler Blockierüberwachung 
	Out_bErrorBlockingMonitoring: BOOL;
END_VAR
VAR_IN_OUT
	/// ISTALosition [mm] 
	InOut_rPosition: REAL;
END_VAR
VAR
	/// interne Variable: Ansteuerung der Achse aktiv 
	bCtrl: BOOL;
	/// interne Variable: Schrittnummer für Schrittkette "Referenzieren mit Referenzschalter" 
	iStepNo: INT;
	/// interne Variable: Steigende Flanke Zählstern 
	rtrigZaehlstern: R_TRIG;
	/// interne Variable: Fallende Flanke Zählstern 
	ftrigZaehlstern: R_TRIG;
	/// interne Variable: Zeitverzögerung Ansteuerung positiv 
	tofCtrlPos: TOF;
	/// interne Variable: Zeitverzögerung Ansteuerung negativ 
	tofCtrlNeg: TOF;
	/// interne Variable: Zeitüberwachung Referenzieren 
	tonBlockingMonitoring: TON;
END_VAR
VAR_INPUT
	/// Achse wird positiv angesteuert 
	In_bCtrlPos: BOOL;
	/// Achse wird positiv angesteuert 
	In_bCtrlNeg: BOOL;
	/// Zählstern auswerten 
	In_bEnable: BOOL;
	/// Eingang des Zählsterns 
	In_bInput: BOOL;
	///Sollwert Position pro Zählstern-Flanke [mm] 
	In_rNominalPositiveEdge: REAL;
	///Sollwert Verzögerung Zählstern auswerten [ms] 
	In_rNominalDelayEvaluation: REAL;
	///Sollwert Verzögerung Blockierüberwachung [ms] 
	In_NominalBlockingDelay: REAL;
	/// Blockierüberwachung nur so lange wie Ansteuerung RDM=FALSE, STAL=TRUE 
	In_bBlockingMonitoringAsLongAsActivation: BOOL := FALSE;
END_VAR

(*******************************************************************************************************************************************)
(* Ansteuerungen verzögern *)
(*******************************************************************************************************************************************)
	(* positive Richtung *)
		tofCtrlPos (IN := In_bCtrlPos, PT:= REAL_TO_TIME(In_rNominalDelayEvaluation));
		
	(* Negative Richtung *)
		tofCtrlNeg (IN := In_bCtrlNeg, PT:= REAL_TO_TIME(In_rNominalDelayEvaluation));
	
	(* Achse wird angesteuert *)
		IF tofCtrlPos.Q OR tofCtrlNeg.Q THEN
			bCtrl:=TRUE;	
		ELSE
			bCtrl:=FALSE;
		END_IF	
			
(*******************************************************************************************************************************************)
(* Flanke bilden *)
(*******************************************************************************************************************************************)
 	(* positive Flankenauswertung Zählstern *)	
		rtrigZaehlstern(CLK:= In_bInput);
	(* Negative Flankenauswertung Zählstern *)	
		ftrigZaehlstern(CLK:= In_bInput);
(*******************************************************************************************************************************************)
(* Position bilden *)
(*******************************************************************************************************************************************)
	(* Zählstern auswerten *)
		IF In_bEnable THEN
			(*Positive Richtung*)
				IF tofCtrlPos.Q AND rtrigZaehlstern.Q THEN
					InOut_rPosition:=InOut_rPosition + In_rNominalPositiveEdge;
				END_IF
			(*Negative Richtung*)
				IF tofCtrlNeg.Q AND ftrigZaehlstern.Q THEN
					InOut_rPosition:=InOut_rPosition - In_rNominalPositiveEdge;
				END_IF
		END_IF
	
(*******************************************************************************************************************************************)
(* Fehlerauswertung *)
(*******************************************************************************************************************************************)
	(* Fehler Blockierüberwachung *)
	(* Achse wird angesteuert und es findet kein Flankenwechsel des Zählsterns statt *)	
	
		IF (In_bBlockingMonitoringAsLongAsActivation = TRUE) THEN
			(* 2014-01-08 Carle: geändert STAL 90 *)(* (bCtrl_pos_i OR bCtrl_neg_i) statt bCtrl *)
			tonBlockingMonitoring(IN := (In_bCtrlPos OR In_bCtrlNeg) AND NOT rtrigZaehlstern.Q AND NOT ftrigZaehlstern.Q,	PT:= REAL_TO_TIME(In_NominalBlockingDelay));		
			IF tonBlockingMonitoring.Q THEN
				Out_bErrorBlockingMonitoring:= TRUE;
			ELSE
				Out_bErrorBlockingMonitoring:= FALSE;
			END_IF
		ELSE
			tonBlockingMonitoring(IN := bCtrl AND	NOT rtrigZaehlstern.Q AND	NOT ftrigZaehlstern.Q, PT:= REAL_TO_TIME(In_NominalBlockingDelay));
		
			IF tonBlockingMonitoring.Q THEN
				Out_bErrorBlockingMonitoring:= TRUE;
			ELSE
				Out_bErrorBlockingMonitoring:= FALSE;
			END_IF
		END_IF

END_FUNCTION_BLOCK

// GeneralFunctionBlocks/FB_ParallelSteps
{attribute 'qualified_only' := ''}
{attribute 'namespace' := 'ILGStdLib.FunctionBlocks'}
FUNCTION_BLOCK FB_ParallelSteps
VAR_OUTPUT
	/// output: Aktueller Schritt aufgrund der "höchswertigsten" Quittierung  
	Out_uiActualStep: UINT;
	/// output: Transition / Weiterschaltung, wenn Einzelschritte beendet oder nicht relevant 
	Out_bTransistion: BOOL;
END_VAR
VAR_IN_OUT
	/// input/output: Status "1" 
	InOut_uiState_01: UINT;
	/// input/output: Status "2" 
	InOut_uiState_02: UINT;
	/// input/output: Status "3" 
	InOut_uiState_03: UINT;
	/// input/output: Status "4" 
	InOut_uiState_04: UINT;
	/// input/output: Status "5" 
	InOut_uiState_05: UINT;
	/// input/output: Status "6" 
	InOut_uiState_06: UINT;
	/// input/output: Status "7" 
	InOut_uiState_07: UINT;
	/// input/output: Status "8" 
	InOut_uiState_08: UINT;
	/// input/output: Status "9" 
	InOut_uiState_09: UINT;
	/// input/output: Status "10" 
	InOut_uiState_10: UINT;
END_VAR
VAR_INPUT
	/// input: Enable: Bausteinbearbeitung 
	In_bEnable: BOOL;
	/// input: Schrittnummer "1" 
	In_uiStep_01: UINT;
	/// input: Schrittnummer "2" 
	In_uiStep_02: UINT;
	/// input: Schrittnummer "3" 
	In_uiStep_03: UINT;
	/// input: Schrittnummer "4" 
	In_uiStep_04: UINT;
	/// input: Schrittnummer "5" 
	In_uiStep_05: UINT;
	/// input: Schrittnummer "6" 
	In_uiStep_06: UINT;
	/// input: Schrittnummer "7" 
	In_uiStep_07: UINT;
	/// input: Schrittnummer "8" 
	In_uiStep_08: UINT;
	/// input: Schrittnummer "9" 
	In_uiStep_09: UINT;
	/// input: Schrittnummer "10" 
	In_uiStep_10: UINT;
	/// input: Schrittnummer für die Transition nach Abarbeitung der Parallelschritte 
	In_uiStepTransition: UINT;
END_VAR

(*==========================================================================================================================================*)
(*		iLLiG_FB_Parallelschritte				    																						*)
(*==========================================================================================================================================*)


(*==========================================================================================================================================*)
(*		Allgemeine Informationen   																				 	 						*)
(*																												    					 	*)
(*																												   							*)
(*		erstellt von:																								 						*)
(*		gt																																 	*)
(*																																 			*)
(*		erforderliche Bibliothek:																								 			*)
(*																													 						*)
(*																													 						*)
(*																													 						*)
(*==========================================================================================================================================*)


(*==========================================================================================================================================*)
(*		Versions-Historie:																							 						*)
(*																												     						*)
(*																												     						*)
(*		17. Januar  	2013	Version 1.0		gt					-	Erstellung						 									*)	
(*																					 											 			*)
(*==========================================================================================================================================*)


(*==========================================================================================================================================*)
(*		Hinweise zur Funktion   																				 				 			*)
(*	Baustein dient zur Ausgabe des aktuellen Status und der aktuellen Schrittnummer bei Parallelschritten.									*)
(*==========================================================================================================================================*)
IF In_bEnable THEN	
	(********************************************************************************************************************************************************)
	(* Ausgabe der aktuellen Schrittnummer aufgrund der "höchstwertigsten Quittierung" **********************************************************************)
	(* Schritt hat Status "1" oder "2" und ist somit aktiv: Ausgabe der Schrittnummer *)
	IF InOut_uiState_01 <> 0
		AND InOut_uiState_01 <> 3
		AND InOut_uiState_01 <> 4 THEN
		Out_uiActualStep := In_uiStep_01;
		Out_bTransistion := FALSE;		
	ELSIF InOut_uiState_02 <> 0
		AND InOut_uiState_02 <> 3
		AND InOut_uiState_02 <> 4 THEN
		Out_uiActualStep := In_uiStep_02;
		Out_bTransistion := FALSE;
	ELSIF InOut_uiState_03 <> 0
		AND InOut_uiState_03 <> 3
		AND InOut_uiState_03 <> 4 THEN
		Out_uiActualStep := In_uiStep_03;
		Out_bTransistion := FALSE;		
	ELSIF InOut_uiState_04 <> 0
		AND InOut_uiState_04 <> 3
		AND InOut_uiState_04 <> 4 THEN
		Out_uiActualStep := In_uiStep_04;
		Out_bTransistion := FALSE;
	ELSIF InOut_uiState_05 <> 0
		AND InOut_uiState_05 <> 3
		AND InOut_uiState_05 <> 4 THEN
		Out_uiActualStep := In_uiStep_05;
		Out_bTransistion := FALSE;
	ELSIF InOut_uiState_06 <> 0
		AND InOut_uiState_06 <> 3
		AND InOut_uiState_06 <> 4 THEN
		Out_uiActualStep := In_uiStep_06;
		Out_bTransistion := FALSE;
	ELSIF InOut_uiState_07 <> 0
		AND InOut_uiState_07 <> 3
		AND InOut_uiState_07 <> 4 THEN
		Out_uiActualStep := In_uiStep_07;
		Out_bTransistion := FALSE;
	ELSIF InOut_uiState_08 <> 0
		AND InOut_uiState_08 <> 3
		AND InOut_uiState_08 <> 4 THEN
		Out_uiActualStep := In_uiStep_08;
		Out_bTransistion := FALSE;
	ELSIF InOut_uiState_09 <> 0
		AND InOut_uiState_09 <> 3
		AND InOut_uiState_09 <> 4 THEN
		Out_uiActualStep := In_uiStep_09;
		Out_bTransistion := FALSE;
	ELSIF InOut_uiState_10 <> 0
		AND InOut_uiState_10 <> 3
		AND InOut_uiState_10 <> 4 THEN
		Out_uiActualStep := In_uiStep_10;
		Out_bTransistion := FALSE;
	ELSE
		(* Transition / Weiterschaltung, wenn Einzelschritte beendet oder nicht relevant ********************************************************************)
		Out_bTransistion := TRUE;		
		Out_uiActualStep := In_uiStepTransition;					(* Schrittnummer für die Transition nach Blockquittierung, wenn also der Block abgearbeitet ist *)				
	END_IF
	(********************************************************************************************************************************************************)
ELSE
	In_uiStep_01					:= 0;								(* input: Schrittnummer "1" *)
	In_uiStep_02					:= 0;								(* input: Schrittnummer "2" *)
	In_uiStep_03					:= 0;								(* input: Schrittnummer "3" *)
	In_uiStep_04					:= 0;								(* input: Schrittnummer "4" *)
	In_uiStep_05					:= 0;								(* input: Schrittnummer "5" *)
	In_uiStep_06					:= 0;								(* input: Schrittnummer "6" *)	
	In_uiStep_07					:= 0;								(* input: Schrittnummer "7" *)
	In_uiStep_08					:= 0;								(* input: Schrittnummer "8" *)
	In_uiStep_09					:= 0;								(* input: Schrittnummer "9" *)
	In_uiStep_10					:= 0;								(* input: Schrittnummer "10" *)	

	InOut_uiState_01				:= 0;								(* input/output: Status "1" *)
	InOut_uiState_02				:= 0;								(* input/output: Status "2" *)
	InOut_uiState_03				:= 0;								(* input/output: Status "3" *)
	InOut_uiState_04				:= 0;								(* input/output: Status "4" *)
	InOut_uiState_05				:= 0;								(* input/output: Status "5" *)
	InOut_uiState_06				:= 0;								(* input/output: Status "6" *)
	InOut_uiState_07				:= 0;								(* input/output: Status "7" *)
	InOut_uiState_08				:= 0;								(* input/output: Status "8" *)
	InOut_uiState_09				:= 0;								(* input/output: Status "9" *)
	InOut_uiState_10				:= 0;								(* input/output: Status "10" *)	

	Out_uiActualStep				:= 0;								(* output: Aktueller Schritt aufgrund der "höchswertigsten" Quittierung  *)
	Out_bTransistion				:= FALSE;							(* output: Transition / Weiterschaltung, wenn Einzelschritte beendet oder nicht relevant *)	
END_IF	
(********************************************************************************************************************************************************)

END_FUNCTION_BLOCK

// GeneralFunctionBlocks/FB_TimeBasedClockGenerator
{attribute 'qualified_only' := ''}
{attribute 'namespace' := 'ILGStdLib.FunctionBlocks'}
FUNCTION_BLOCK FB_TimeBasedClockGenerator
VAR_IN_OUT
	/// output: Zeitbasierter Taktgeber
	InOut_bClock: BOOL;
END_VAR
VAR
	/// lokale Variable: Initialisierung ist erfolgt. Damit der Baustein sofrt nach der Initialisierung bereit ist, auch wenn bEnable_in statisch "TRUE" ist *)	(* 2012-02-14 gt: hinzu *)
	bInit: BOOL;
	/// lokale Variable: Startsignal ist erfolgt, ab jetzt wird der Takt ausgegeben
	bStartSignal: BOOL;
	/// lokale Variable: Vorgegebener Zeitwert im TIME-Format: Für Zeitglied 1
	tTimeValueTimer1: TIME;
	/// lokale Variable: Vorgegebener Zeitwert im TIME-Format: Für Zeitglied 2
	tTimeValueTimer2: TIME;
	/// lokale Variable: Takt-Impuls des Startsignals bilden
	rtrigStartPulse: R_TRIG;
	/// lokale Variable: Impuls: Starten des Taktgebers
	bStartPulse: BOOL;
	/// lokale Variable: Zeitglied 1 hat aktuellen Zeitwert
	bTimeReachedTimer1: BOOL;
	/// lokale Variable: Zeitglied 2 hat aktuellen Zeitwert
	bTimeReachedTimer2: BOOL;
	/// lokale Variable: Zeitglied 1 für die Taktvorgabe
	tonTimer1: TON;
	/// lokale Variable: Zeitglied 2 für die Taktvorgabe
	tonTimer2: TON;
END_VAR
VAR_INPUT
	/// input: Solange der "bEnable" nicht "TRUE" ist, erfolgt keine Auswertung
	In_bEnable: BOOL;
	/// input: Start des zeitbasierten Taktgebers
	In_bStart: BOOL;
	/// [ms] Zeitwert für den Taktgeber
	In_rTimeValueClockGenerator_ms: REAL;
END_VAR

// Impuls bei Takt bilden ===============================================================================================================
rtrigStartPulse(CLK:= In_bStart , Q=> );

// Impuls als BOOLsche Variable =========================================================================================================
bStartPulse := rtrigStartPulse.Q;

// Startsignal ist erfolgt, ab jetzt wird der Takt ausgegeben ===========================================================================
IF In_bEnable AND bStartPulse THEN
	bStartSignal := TRUE;  						
END_IF

// Zeitwert REAL --> TIME-Format ========================================================================================================
IF NOT tonTimer1.IN THEN
	tTimeValueTimer1 := REAL_TO_TIME(In_rTimeValueClockGenerator_ms);
END_IF
IF NOT tonTimer2.IN THEN
	tTimeValueTimer2 := REAL_TO_TIME(In_rTimeValueClockGenerator_ms);
END_IF
//=======================================================================================================================================
IF In_bEnable AND bInit THEN
	// Zeitglied 1 ======================================================================================================================	
	tonTimer1(	IN :=	bTimeReachedTimer1 AND	
						(bStartSignal OR tonTimer1.IN		// Selbsthaltung
						)
						AND NOT tonTimer1.Q	
						AND NOT tonTimer2.IN,			// Das andere Zeitglied ist NICHT aktiv
						PT := tTimeValueTimer1
			  );

	bTimeReachedTimer2	:= 	(	NOT bTimeReachedTimer1
								AND NOT tonTimer1.Q
							)
							OR	(	tonTimer2.IN
									AND NOT tonTimer2.Q
								)
							OR	(	tonTimer1.Q
									AND NOT tonTimer2.Q
									//AND NOT FB_Zeitglied_1_TON_Takt_Takt_lokal.IN
								);								
	
	// Zeitglied 2 ======================================================================================================================	
	tonTimer2	( 	IN := 	bTimeReachedTimer2
							AND	(	bStartSignal
									OR tonTimer2.IN		// Selbsthaltung
								)
							AND NOT tonTimer1.IN,			// Das andere Zeitglied ist NICHT aktiv
					PT := tTimeValueTimer2
				);

	bTimeReachedTimer1 :=	(	NOT bTimeReachedTimer2
								AND NOT tonTimer2.Q
							)
							OR	(	tonTimer1.IN
									AND NOT tonTimer1.Q
								)
							OR	(	tonTimer2.Q
									AND NOT tonTimer1.Q
									//AND NOT FB_Zeitglied_2_TON_Takt_Takt_lokal.IN
								);
										
ELSE
	bStartSignal := FALSE;  						
	bTimeReachedTimer1 := TRUE;
	bTimeReachedTimer2 := FALSE;	
	tonTimer1.IN := FALSE;
	tonTimer2.IN := FALSE;
	bInit := TRUE;
END_IF
//=======================================================================================================================================
// Ausgabe: Zeitbasierter Taktgeber
InOut_bClock := tonTimer1.Q	OR tonTimer2.Q;
//=======================================================================================================================================

END_FUNCTION_BLOCK

// GeneralFunctionBlocks/FB_TriggerValueChange
{attribute 'qualified_only' := ''}
{attribute 'namespace' := 'ILGStdLib.FunctionBlocks'}
FUNCTION_BLOCK FB_TriggerValueChange
VAR_OUTPUT
	OUT_bTrigger: BOOL;
END_VAR
VAR
	rValue1Old: REAL;
	rValue2Old: REAL;
	rValue3Old: REAL;
	rValue4Old: REAL;
	rValue5Old: REAL;
	rValue6Old: REAL;
	rValue7Old: REAL;
	rValue8Old: REAL;
	rValue9Old: REAL;
	rValue10Old: REAL;
	rValue11Old: REAL;
	rValue12Old: REAL;
	rValue13Old: REAL;
	rValue14Old: REAL;
	rValue15Old: REAL;
	rValue16Old: REAL;
	rValue17Old: REAL;
	rValue18Old: REAL;
	rValue19Old: REAL;
	rValue20Old: REAL;
	rValue21Old: REAL;
	rValue22Old: REAL;
	rValue23Old: REAL;
	rValue24Old: REAL;
	rValue25Old: REAL;
	rValue26Old: REAL;
	rValue27Old: REAL;
	rValue28Old: REAL;
	rValue29Old: REAL;
	rValue30Old: REAL;
	rValue31Old: REAL;
	rValue32Old: REAL;
	rValue33Old: REAL;
	rValue34Old: REAL;
	rValue35Old: REAL;
	rValue36Old: REAL;
	rValue37Old: REAL;
	rValue38Old: REAL;
	rValue39Old: REAL;
	rValue40Old: REAL;
	bTriggerOld: BOOL;
END_VAR
VAR_INPUT
	In_bEnable: BOOL;
	In_rValue1: REAL := 0.0;
	In_rValue2: REAL := 0.0;
	In_rValue3: REAL := 0.0;
	In_rValue4: REAL := 0.0;
	In_rValue5: REAL := 0.0;
	In_rValue6: REAL := 0.0;
	In_rValue7: REAL := 0.0;
	In_rValue8: REAL := 0.0;
	In_rValue9: REAL := 0.0;
	In_rValue10: REAL := 0.0;
	In_rValue11: REAL := 0.0;
	In_rValue12: REAL := 0.0;
	In_rValue13: REAL := 0.0;
	In_rValue14: REAL := 0.0;
	In_rValue15: REAL := 0.0;
	In_rValue16: REAL := 0.0;
	In_rValue17: REAL := 0.0;
	In_rValue18: REAL := 0.0;
	In_rValue19: REAL := 0.0;
	In_rValue20: REAL := 0.0;
	In_rValue21: REAL := 0.0;
	In_rValue22: REAL := 0.0;
	In_rValue23: REAL := 0.0;
	In_rValue24: REAL := 0.0;
	In_rValue25: REAL := 0.0;
	In_rValue26: REAL := 0.0;
	In_rValue27: REAL := 0.0;
	In_rValue28: REAL := 0.0;
	In_rValue29: REAL := 0.0;
	In_rValue30: REAL := 0.0;
	In_rValue31: REAL := 0.0;
	In_rValue32: REAL := 0.0;
	In_rValue33: REAL := 0.0;
	In_rValue34: REAL := 0.0;
	In_rValue35: REAL := 0.0;
	In_rValue36: REAL := 0.0;
	In_rValue37: REAL := 0.0;
	In_rValue38: REAL := 0.0;
	In_rValue39: REAL := 0.0;
	In_rValue40: REAL := 0.0;
END_VAR

IF NOT bTriggerOld THEN
	OUT_bTrigger := FALSE;

	IF NOT In_bEnable THEN

		OUT_bTrigger := FALSE;
	
	ELSE
		IF (In_rValue1 <> rValue1Old) THEN
			OUT_bTrigger := TRUE;
			rValue1Old := In_rValue1;
		END_IF
	
		IF (In_rValue2 <> rValue2Old)  THEN
			OUT_bTrigger := TRUE;
			rValue2Old := In_rValue2;
		END_IF
	
		IF (In_rValue3 <> rValue3Old)  THEN
			OUT_bTrigger := TRUE;
			rValue3Old := In_rValue3;
		END_IF
	
		IF (In_rValue4 <> rValue4Old)  THEN
			OUT_bTrigger := TRUE;
			rValue4Old := In_rValue4;
		END_IF
	
		IF (In_rValue5 <> rValue5Old)  THEN
			OUT_bTrigger := TRUE;
			rValue5Old := In_rValue5;
		END_IF
	
		IF (In_rValue6 <> rValue6Old)  THEN
			OUT_bTrigger := TRUE;
			rValue6Old := In_rValue6;
		END_IF
	
	
		IF (In_rValue7 <> rValue7Old)  THEN
			OUT_bTrigger := TRUE;
			rValue7Old := In_rValue7;
		END_IF
	
	
		IF (In_rValue8 <> rValue8Old)  THEN
			OUT_bTrigger := TRUE;
			rValue8Old := In_rValue8;
		END_IF
	
	
		IF (In_rValue9 <> rValue9Old)  THEN
			OUT_bTrigger := TRUE;
			rValue9Old := In_rValue9;
		END_IF
	
	
		IF (In_rValue10 <> rValue10Old)  THEN
			OUT_bTrigger := TRUE;
			rValue10Old := In_rValue10;
		END_IF
	
		IF (In_rValue11 <> rValue11Old)  THEN
			OUT_bTrigger := TRUE;
			rValue11Old := In_rValue11;
		END_IF
	
		IF (In_rValue12 <> rValue12Old)  THEN
			OUT_bTrigger := TRUE;
			rValue12Old := In_rValue12;
		END_IF
	
		IF (In_rValue13 <> rValue13Old)  THEN
			OUT_bTrigger := TRUE;
			rValue13Old := In_rValue13;
		END_IF
	
		IF (In_rValue14 <> rValue14Old)  THEN
			OUT_bTrigger := TRUE;
			rValue14Old := In_rValue14;
		END_IF
	
		IF (In_rValue15 <> rValue15Old)  THEN
			OUT_bTrigger := TRUE;
			rValue15Old := In_rValue15;
		END_IF
	
		IF (In_rValue16 <> rValue16Old)  THEN
			OUT_bTrigger := TRUE;
			rValue16Old := In_rValue16;
		END_IF
	
		IF (In_rValue17 <> rValue17Old)  THEN
			OUT_bTrigger := TRUE;
			rValue17Old := In_rValue17;
		END_IF

		IF (In_rValue18 <> rValue18Old)  THEN
			OUT_bTrigger := TRUE;
			rValue18Old := In_rValue18;
		END_IF

		IF (In_rValue19 <> rValue19Old)  THEN
			OUT_bTrigger := TRUE;
			rValue19Old := In_rValue19;
		END_IF

		IF (In_rValue20 <> rValue20Old)  THEN
			OUT_bTrigger := TRUE;
			rValue20Old := In_rValue20;
		END_IF

		IF (In_rValue21 <> rValue21Old)  THEN
			OUT_bTrigger := TRUE;
			rValue21Old := In_rValue21;
		END_IF

		IF (In_rValue22 <> rValue22Old)  THEN
			OUT_bTrigger := TRUE;
			rValue22Old := In_rValue22;
		END_IF

		IF (In_rValue23 <> rValue23Old)  THEN
			OUT_bTrigger := TRUE;
			rValue23Old := In_rValue23;
		END_IF

		IF (In_rValue24 <> rValue24Old)  THEN
			OUT_bTrigger := TRUE;
			rValue24Old := In_rValue24;
		END_IF

		IF (In_rValue25 <> rValue25Old)  THEN
			OUT_bTrigger := TRUE;
			rValue25Old := In_rValue25;
		END_IF

		IF (In_rValue26 <> rValue26Old)  THEN
			OUT_bTrigger := TRUE;
			rValue26Old := In_rValue26;
		END_IF

		IF (In_rValue27 <> rValue27Old)  THEN
			OUT_bTrigger := TRUE;
			rValue27Old := In_rValue27;
		END_IF

		IF (In_rValue28 <> rValue28Old)  THEN
			OUT_bTrigger := TRUE;
			rValue28Old := In_rValue28;
		END_IF

		IF (In_rValue29 <> rValue29Old)  THEN
			OUT_bTrigger := TRUE;
			rValue29Old := In_rValue29;
		END_IF

		IF (In_rValue30 <> rValue30Old)  THEN
			OUT_bTrigger := TRUE;
			rValue30Old := In_rValue30;
		END_IF

		IF (In_rValue31 <> rValue31Old)  THEN
			OUT_bTrigger := TRUE;
			rValue31Old := In_rValue31;
		END_IF

		IF (In_rValue32 <> rValue32Old)  THEN
			OUT_bTrigger := TRUE;
			rValue32Old := In_rValue32;
		END_IF

		IF (In_rValue33 <> rValue33Old)  THEN
			OUT_bTrigger := TRUE;
			rValue33Old := In_rValue33;
		END_IF

		IF (In_rValue34 <> rValue34Old)  THEN
			OUT_bTrigger := TRUE;
			rValue34Old := In_rValue34;
		END_IF

		IF (In_rValue35 <> rValue35Old)  THEN
			OUT_bTrigger := TRUE;
			rValue35Old := In_rValue35;
		END_IF

		IF (In_rValue36 <> rValue36Old)  THEN
			OUT_bTrigger := TRUE;
			rValue36Old := In_rValue36;
		END_IF

		IF (In_rValue37 <> rValue37Old)  THEN
			OUT_bTrigger := TRUE;
			rValue37Old := In_rValue37;
		END_IF

		IF (In_rValue38 <> rValue38Old)  THEN
			OUT_bTrigger := TRUE;
			rValue38Old := In_rValue38;
		END_IF

		IF (In_rValue39 <> rValue39Old)  THEN
			OUT_bTrigger := TRUE;
			rValue39Old := In_rValue39;
		END_IF

		IF (In_rValue40 <> rValue40Old)  THEN
			OUT_bTrigger := TRUE;
			rValue40Old := In_rValue40;
		END_IF

	END_IF

ELSE
	OUT_bTrigger := FALSE;

END_IF


bTriggerOld := OUT_bTrigger;

END_FUNCTION_BLOCK

// GeneralFunctionBlocks/FB_ValueIsIntegerMultiple
{attribute 'qualified_only' := ''}
{attribute 'namespace' := 'ILGStdLib.FunctionBlocks'}
FUNCTION_BLOCK FB_ValueIsIntegerMultiple
VAR_OUTPUT
	/// Zu prüfender Wert ist ein ganzzahliges Vielfaches
	Out_bIsIntegerMultiple: BOOL;
	/// Vorkomma-Teil der Differenz: Nachkomma abschneiden
	Out_uiBeforeCommaPart: UINT;
	/// Nachkomma-Teil der Differenz = Differenz - Vorkomma-Teil
	Out_rAfterCommaPart: REAL;
END_VAR
VAR
	/// Differenz: rZu_pruefender_Wert_in / rDivisor_in
	rDifference: REAL;
	/// Steigende Flanke "Nachkomma-Teil ist gleich 0000"
	rtrigAfterCommaPartIsNull: R_TRIG;
END_VAR
VAR_INPUT
	/// Bausteinbearbeitung, wenn TRUE
	In_bEnable: BOOL;
	/// Wert, der auf Ganzzahliges Vielfaches geprüft werden soll (Real-Wert mit EINER Nachkommastelle)
	In_rValueToCheck: REAL;
	/// Divisor (Nenner), durch den der "rZu_pruefender_Wert_in" geteilt wird	
	In_rDivisor: REAL;
END_VAR

IF In_bEnable THEN
	// Ist der "rZu_pruefender_Wert_in" ein ganzzahliges Vielfaches von "rDivisor_in", wird der Ausgang
	// "bGanzzahliges_Vielfaches_out" ausgegeben.
	// Beispiel:	"rDivisor_in" ist 80.0 und somit wird der Ausgang "bGanzzahliges_Vielfaches_out" bei
	// 				rZu_pruefender_Wert_in = 80.0, 160.0, 240.0, 320, also n*80.0 ausgegeben
	rDifference := F_lrRound((In_rValueToCheck / In_rDivisor), 2);
	Out_uiBeforeCommaPart := DINT_TO_UINT(TRUNC(rDifference));									// Vorkomma-Teil der Differenz: Nachkomma abschneiden
	Out_rAfterCommaPart := F_lrRound((rDifference - UINT_TO_REAL(Out_uiBeforeCommaPart)), 2);	// Nachkomma-Teil der Differenz = Differenz - Vorkomma-Teil
	
	rtrigAfterCommaPartIsNull(CLK:= (Out_rAfterCommaPart = 0.000));					// Steigende Flanke "Nachkomma-Wert ist gleich 0000"
	
	// Wenn Schmierimpuls = 80, 160, 240, 320,...800 dann Zyklus inkrementieren
	IF (rDifference > 0.0)
		AND rtrigAfterCommaPartIsNull.Q THEN
		Out_bIsIntegerMultiple := TRUE;														// Zu prüfender Wert ist ein ganzzahliges Vielfaches
	ELSE
		Out_bIsIntegerMultiple := FALSE;														// Zu prüfender Wert ist ein ganzzahliges Vielfaches
	END_IF	
ELSE
	Out_bIsIntegerMultiple := FALSE;															// Zu prüfender Wert ist ein ganzzahliges Vielfaches
	Out_uiBeforeCommaPart := 0;																		// Vorkomma-Teil der Differenz: Nachkomma abschneiden
	Out_rAfterCommaPart := 0.0;																		// Nachkomma-Teil der Differenz = Differenz - Vorkomma-Teil
END_IF

END_FUNCTION_BLOCK

// GeneralFunctions/Math/F_lrRound
{attribute 'qualified_only' := ''}
{attribute 'namespace' := 'ILGStdLib.Functions.Math'}
FUNCTION F_lrRound : LREAL
VAR_INPUT
	In_rValue: REAL;
	In_iDigits: INT;
END_VAR
VAR
	diValueTrunc: DINT;
	rValueRest: REAL;
	rValueTemp: REAL;
END_VAR

rValueTemp:=LREAL_TO_REAL(In_rValue * EXPT(10,In_iDigits));

diValueTrunc := TRUNC_INT(rValueTemp);
rValueRest := rValueTemp - DINT_TO_REAL(diValueTrunc);

IF rValueRest < 0.5 THEN
	F_lrRound := DINT_TO_REAL(diValueTrunc) / EXPT(10,In_iDigits);
ELSE
	F_lrRound := DINT_TO_REAL(diValueTrunc+1) / EXPT(10,In_iDigits);
END_IF

END_FUNCTION

// GeneralFunctionBlocks/FB_VIMP
{attribute 'qualified_only' := ''}
{attribute 'namespace' := 'ILGStdLib.FunctionBlocks'}
FUNCTION_BLOCK FB_VIMP
VAR_OUTPUT
	/// Timer läuft 
	Out_bTimerRunning: BOOL;
END_VAR
VAR
	/// Start speichern 
	bStartStored: BOOL;
	/// Steigende Flanke Start 
	rtrigStart: R_TRIG;
	/// Einschaltverzögerung Start 
	tonStart: TON;
END_VAR
VAR_INPUT
	/// Start Timer 
	In_bStart: BOOL;
	/// Impulszeit [ms]
	In_rSWTime: REAL;
END_VAR


(* Positve Flanke des Eingangsignal "Start" bilden *)
rtrigStart(CLK:= In_bStart);
(* Start rücksetzen *)
IF (bStartStored AND rtrigStart.Q) OR tonStart.Q THEN
	bStartStored := FALSE;
END_IF
(* Start speichern *)
IF (NOT bStartStored AND rtrigStart.Q) THEN
	bStartStored := TRUE;
END_IF

(* Einschaltverzögerung des Startsignals *)
tonStart(IN := bStartStored, PT:= REAL_TO_TIME(In_rSWTime));
	
(* Ausgang setzen, solange Timer läuft *)
Out_bTimerRunning := bStartStored AND NOT tonStart.Q;

END_FUNCTION_BLOCK

// InternalFunctions/FUN_WriteLnString
FUNCTION FUN_WriteLnString : UDINT
VAR_INPUT
	/// file handle 
	hHandle: ITF_FILEASYNC;
	/// argument for format string 
	sArg: STRING(255);
END_VAR
VAR
	/// format string 
	// fb_FileWriteAsyc: IL_FileWriteAsync;	
	sFormat: STRING(20) := '%s$R$N';
	udiBytesWritten : UDINT;	
END_VAR

// FUN_WriteLnString := SysFileStreamFPrintf_String(dwHandle, sFormat, ADR(sArg));
(* Funktioniert so nicht, da kein FB in Funktion verwendet werden darf !!!
fb_FileWriteAsyc(
	Execute:= TRUE,
	BufferAddr=> ,
	BufferSize=> ,
	FileHandle:= hHandle,
	Done=> ,
	Active=> ,
	Error=> ,
	ErrorId=> ,
	ErrorIdent=> ,
	BytesWritten=> udiBytesWritten);


IF IL_FileWriteAsync.Done THEN
	
END_IF
*)
FUN_WriteLnString := udiBytesWritten;

END_FUNCTION

// GeneralFunctionBlocks/ActivateDevices/FB_ActivateDevices
///Program ActivateDevices
/// 	
///	                                 ******************
///                                     *   DISCLAIMER   *
///                                     ******************
///   It is acknowledged that with regard to these software programs and program modules free of
///   charge, Bosch Rexroth's usually practised, in-house test and release procedures have not 
///   been accomplished. These software programs and program modules free of charge serve only as
///   an example for possible applications.  They are intended as a help in order to obtain addi-
///   tional experience regarding function, operation, performance and capacity of a maybe later 
///   issued series release. Therefore Bosch Rexroth disclaims any liability and rejects to assume
///   responsibility that these software programs or program modules, including any information 
///   and data stored in those programs, are suitable for any intended use or that these programs
///   will work without errors in any combination with the data processing environment. Providing 
///   you with these software programs shall neither constitute a claim for technical support nor
///   for any other remedy for defects. Any claims for damages of any nature and for any legal
///   reason arising from installing or using these software programs or program modules are ex-
///   cluded, unless these damages was caused by Bosch Rexroth`s statutory representatives or em-
///   ployees by wilful misconduct or by gross negligence or liability is compulsory in accordance
///   with the German product liability law. In any case Bosch Rexroth`s liability for any conse-
///   quential or incidental damages such as, but not limited to loss of profit, loss of pro-
///   duction or loss of data is excluded.      
///
///##############################################################################################
///##############################################################################################
///
///General Header
///----------------------------------------------------------------------------------------------
///Short description      : active and passive handling for drives, sercos IO, PN IO 
///						 and local S20 IO with XM control
///Version                : 14.8.XM
///Author                 : Jörg Schneider
///Date                   : 2019-10-24 
///Company                : DC-AE/STS2
///Target                 : MLC 14VRS
///----------------------------------------------------------------------------------------------
/// Additional Header 																			
///----------------------------------------------------------------------------------------------
/// Used Libraries 																				
///		- Util.library																			
///		- SysFileAsync23.library																
///		- SysDir.library																		
///		- CmpErrors.library																		
///		- SysTypes.library																		
///		- ML_TechBase.library 																	
///      - RIL_Inline.library																	
///      - RIL_InlineIOModules.library															
///      - RIH_IndraControl_S20.library															
///##############################################################################################
///##############################################################################################
///		Possible Errors 																		
///																								
///		ERROR_CODE			ERROR_TABLE		Add1		Add2		Description					
///----------------------------------------------------------------------------------------------
///		RESOURCE_ERROR		USER1_TABLE		16#F0001	16#F0000	difference between found 	
///																												and configured drives.		
///																												See Output DeviceConfigError.Axes	
///																								
///		RESOURCE_ERROR		USER1_TABLE		16#F0002	16#F0000	drive found which is not in 
///																												C-0-0478 					
///																												See Output DeviceConfigError.FoundDrives	
///																								
///		RESOURCE_ERROR		USER1_TABLE		16#F0003	16#F0000	Error in sercos IO configuration 
///																												See Output DeviceConfigError.sercos_IO	
///																								
///		RESOURCE_ERROR		USER1_TABLE		16#F0004	16#F0000	Error in sercos IO configuration 
///																												See Output DeviceConfigError.sercos_IO_CmdConfig	
///																								
///----------------------------------------------------------------------------------------------
/// History			 																			
///----------------------------------------------------------------------------------------------
/// Version:		14.1.0 																			
/// Date: 		2016-10-17																		
/// Name: 		Jörg Schneider (DC-IA/SDF61) 													
/// Comment:		First Release for MLC 14														
/// 					 																			
/// 					 																			
/// Version:		14.2.0 																			
/// Date: 		2017-02-27																		
/// Name: 		Jörg Schneider (DC-IA/SDF61) 													
/// Comment:		Include replacement for UIL_StringHandling.library								
/// 					 																			
/// 					 																			
/// Version:		14.3.0 																			
/// Date: 		2017-12-06																		
/// Name: 		Jörg Schneider (DC-IA/SDF61) 													
/// Comment:		remove UIL_StringHandlingReplacement 											
/// 					 																			
/// 					 																			
/// Version:		14.4.0 																			
/// Date: 		2018-02-21																		
/// Name: 		Jürgen Kohl (DC-AE/STS2) 														
/// Comment:		In state 40:																	
///				"IF udiNoOfElements2 > 7 THEN" replaced with "IF udiNoOfElements > 7 THEN"		
///				In state 290:																	
///				additional Concat sequence inserted to get the whole error message				
/// 					 																			
/// 					 																			
/// Version:		14.5.XM																			
/// Date: 		2019-03-05																		
/// Name: 		Jörg Schneider (DC-AE/STS2) 													
/// Comment:		remove inline, PROFINET and sercos i/o handling for XM control					
/// 					 																			
/// 					 																			
/// Version:		14.6.XM																			
/// Date: 		2019-03-12																		
/// Name: 		Jörg Schneider (DC-AE/STS2) 													
/// Comment:		add sercos i/o handling for XM control											
/// 				remove SysFileStream23.library													
/// 					 																			
/// Version:		14.7.XM																			
/// Date: 		2019-03-25																		
/// Name: 		Jörg Schneider (DC-AE/STS2) 													
/// Comment:		add EFC FUN_TypeCodeIsRexrothIO													
/// 				change get TypeCode of sercos IO in step 40 									
/// 					 																			
/// Version:		14.8.XM																			
/// Date: 		2019-11-15																		
/// Name: 		Jörg Schneider (DC-AE/STS2) 													
/// Comment:		add local S20 IO handling														
/// 				add PN IO handling							 									
/// 				extend DUT_S20Type							 									
/// 					 																			
/// Former Programm, now FB to get it into a library                                             
/// Date: 04.04.2025                                                                             
/// Name: Dirk Süß                                                                               
///                                                                                              
FUNCTION_BLOCK FB_ActivateDevices IMPLEMENTS ITF_ActivateDevices
VAR_OUTPUT
	/// FB is active
	OUT_bActive: BOOL;
	/// FB is finished
	OUT_bDone: BOOL;
	/// FB has an Error
	OUT_bError: BOOL;
	/// Reboot of MLC required
	OUT_bReboot: BOOL;
	OUT_ErrorID: ERROR_CODE;
	OUT_ErrorIdent: ERROR_STRUCT;
	/// First Error is described in Message 	
	OUT_sDiagMessage: STRING(255);
END_VAR
VAR
	/// Update Drive fimrware and Functional Package if needed
	bUpdateFirmware: BOOL := FALSE;
	refastAxesCmdConfig: REFERENCE TO ARRAY [1..iMAX_AXES_NUMBER] OF ST_AxesCmdConfig;
	refastInlineIOCmdConfig: REFERENCE TO ARRAY [1..iMAX_S20_IO] OF ST_InlineIOCmdConfig;
	refastSercosIOCmdConfig: REFERENCE TO ARRAY [1..iMAX_SERCOS_IO] OF ST_SercosIOCmdConfig;
	refastProfibusIOCmdConfig: REFERENCE TO ARRAY [1..iMAX_PROFIBUS_MASTER, 0..iMAX_PROFIBUS_SLAVE] OF ST_ProfibusIOCmdConfig;
	refastPNIOCmdConfig: REFERENCE TO ARRAY [1..iMAX_PN_MASTER, 0..iMAX_PN_SLAVE] OF ST_PNIOCmdConfig;
	refastAxesActConfig: REFERENCE TO ARRAY [1..iMAX_AXES_NUMBER] OF ST_AxesActConfig;
	refastInlineIOActConfig: REFERENCE TO ARRAY [1..iMAX_INLINE_IO] OF ST_InlineIOActConfig;
	refastSercosIOActConfig: REFERENCE TO ARRAY [1..iMAX_SERCOS_IO] OF ST_SercosIOActConfig;
	refastSercosIOActConfigC578: ARRAY[1..iMAX_SERCOS_IO] OF ST_SercosIOActConfig;
	///	PNIOActConfig :REFERENCE TO ARRAY [1..MAX_PN_MASTER,1..MAX_PN_SLAVE] OF DUT_PNIOActConfig;
	refastAxesConfigError: REFERENCE TO ARRAY [1..iMAX_AXES_NUMBER] OF ST_AxesConfigError;
	refastSercosIOConfigError: REFERENCE TO ARRAY [1..iMAX_SERCOS_IO] OF ST_SercosIOConfigError;
	///	SercosIOCmdConfigError		: REFERENCE TO DUT_SercosIOCmdConfigError;
	refastInlineIOConfigError: REFERENCE TO ARRAY [1..iMAX_INLINE_IO] OF ST_InlineIOConfigError;
	refastFoundDrivesError: REFERENCE TO ARRAY [1..iMAX_AXES_NUMBER] OF ST_AxesConfigErrorFoundDrives;
	stDummyAxesActConfig: ST_AxesActConfig;
	astAxesActConfigTmp: ARRAY[1..iMAX_AXES_NUMBER] OF ST_AxesActConfig;
	astSercosIOActConfigTmp: ARRAY[1..iMAX_SERCOS_IO] OF ST_SercosIOActConfig;
	bExecuteOld: BOOL;
	bErrorTemp: BOOL;
	{ warning '###TODO: Für Sercos, muss in ctrlX auf Ethercat umgebaut werden' }
	(* Für Sercos, muss in ctrlX auf Ethercat umgebaut werden
	fbCommand: MB_Command;
	fbReadListParameter: MB_ReadListParameter;
	fbWriteListParameter: MB_WriteListParameter;
	fbWriteA24: MB_WriteParameter;
	*)
	stDummyAxis: AXIS_REF;
	iState: INT;
	iA24: INT;
	i: INT;
	j: INT;
	k: INT;
	l: INT;
	m: INT;
	uiLengthArC510: UINT;
	aiC484: ARRAY[1..(2 * iMAX_AXES_NUMBER)] OF INT;
	aiC510: ARRAY[1..iMAX_SERCOS_DEVICES] OF INT;
	apiPointerToC510: ARRAY[1..iMAX_SERCOS_DEVICES] OF POINTER TO INT;
	sRingString: STRING((100 * iMAX_SERCOS_DEVICES));
	sC578: STRING((100 * iMAX_SERCOS_DEVICES));
	sRingString2: STRING((100 * iMAX_SERCOS_DEVICES));
	sTemp: STRING(20);
	psString: POINTER TO STRING;
	psRingString2: POINTER TO STRING(120);
	psStringTemp: POINTER TO STRING;
	/// array of all axis elements
	apsElements: ARRAY[1..(iMAX_SERCOS_DEVICES * iMAX_NUM_ELEMENTS_C479)] OF POINTER TO STRING(255);
	///Temp string to prepare elements
	apsElements2: ARRAY[1..20] OF POINTER TO STRING(255);
	/// array of all axis elements
	apsSplit: ARRAY[1..(iMAX_SERCOS_DEVICES * iMAX_NUM_ELEMENTS_C479)] OF POINTER TO STRING(255);
	asAxisString: ARRAY[1..iMAX_SERCOS_DEVICES] OF STRING;
	pbByteTemp: POINTER TO BYTE;
	pbByteTemp2: POINTER TO BYTE;
	/// Add FB
	fbReadStringParameter: MB_ReadStringParameter;
	/// TODO: Add FB
	WriteC578: MB_WriteListParameter;
	bExecuteReadName: BOOL;
	sTemp1: STRING;
	sTemp2: STRING;
	sTemp3: STRING;
	sComma: STRING;
	sSercosAdress: STRING;
	sDiagMessageInt: STRING(255);
	iSercosAddressTemp: INT;
	iActConfigInlineIO: INT;
	iActNoOfDrives: INT;
	iActNoOfSercosIO: INT;
	iLineCfg: INT;
	asStringCmdCfg: ARRAY[1..iMAX_LINE_CFG] OF STRING(80);
	asStringActCfg: ARRAY[1..iMAX_LINE_CFG] OF STRING(80);
	fb_SysFileOpenAsync: SysFileOpenAsync;
	hCfg: DWORD;
	sBuffer: STRING(iMAX_BUFFER_SIZE);
	fb_SysFileReadAsync: SysFileReadAsync;
	fb_SysFileCloseAsync: SysFileCloseAsync;
	iFileSize: INT := iMAX_BUFFER_SIZE;
	dwReadBytes: DWORD;
	sLineFeed: STRING(1);
	sLineFeed2: STRING(2);
	bExecuteWriteA24: BOOL;
	iEOF: INT;
	diResult: DINT;
	astDirEntry: ARRAY[0..iMAX_DIR_ENTRY] OF ST_DirEntry;
	iEntry: INT;
	diMaxEntry: DINT;
	dir: DirInfo;
	Result: RTS_IEC_RESULT;
	hDir: RTS_IEC_HANDLE;
	bLoopend: BOOL;
	fbINLNModuleConfigList: IL_INLNModuleConfigList;
	InlineIOCfg: ARRAY[1..iMAX_INLINE_IO] OF IL_INLINE_CFG_ID_DESC;
	udiNoOfModuleConfig: UDINT;
	sPathNameInt: STRING := sPATH_NAME;
	sFileAndPathInt: STRING := sFILE_AND_PATH;
	/// Read Serial
	bExecuteReadSerialNo: BOOL;
	audiP1518: ARRAY[0..7] OF UDINT;
	/// Read SafetyType
	bExecuteReadSafetyType: BOOL;
	/// Read S20 ModuleType
	bExecuteReadModuleType: BOOL;
	aliS1500_0_3: ARRAY[0..63] OF LINT;
	bWriteThisLine: BOOL;
	/// Variable for Read Fimware Directory
	///--------------------------------------
	sTemp4: STRING;
	astDirInfo: ARRAY[1..99] OF DirInfo;
	udiResultOpen: UDINT;
	///	ar_sFirmwareFiles 			: ARRAY [1..MAX_NO_FIRMWARE_FILES] OF STRING(99);	
	///	ar_stFirmwareFilesType 		: ARRAY [1..MAX_NO_FIRMWARE_FILES] OF DUT_FirmwareType;	
	///	sFirmwareDirectoryTemp		: STRING := '/ata0b/DriveFirmware';
	///	udiDirHandle: RTS_IEC_HANDLE;
	///	uiNoOfFimrwareFiles : UINT;
	uiFileNo: UINT;
	udiResultRead: RTS_IEC_RESULT;
	stActFirmwareType: ST_FirmwareType;
	ar_bFirmwareUpdate: ARRAY[1..iMAX_AXES_NUMBER] OF BOOL;
	ar_uiUpdateFileNo: ARRAY[1..iMAX_AXES_NUMBER] OF UINT := [iMAX_AXES_NUMBER(1)];
	uiNoOfFirmwareFiles: UINT;
	stCmdFirmwareType: ST_FirmwareType;
	///	fbTFTPPutFileAsync: ARRAY[1..MAX_AXES_NUMBER] OF IL_TFTPPutFileAsync;
	afbWriteP2003: ARRAY[1..iMAX_AXES_NUMBER] OF MB_WriteParameter;
	abDriveIP: ARRAY[0..3] OF BYTE;
	bScanAgain: BOOL;
	abWriteP2003: ARRAY[1..iMAX_AXES_NUMBER] OF BOOL;
	bRebootDrive: BOOL;
	fbCommandRebootDrive: ARRAY[1..iMAX_AXES_NUMBER] OF MB_Command;
	fbWaitReboot: TON;
	iP2003: INT;
	///fbReset: ARRAY[1..MAX_AXES_NUMBER] OF MC_Reset;
	fbResetMLC: MC_Reset;
	wTemp: WORD;
	fbWriteC506: MB_WriteParameter;
	udiResutlCreate: RTS_IEC_RESULT;
	dwC506: DWORD;
	bIOFound: BOOL;
	abSercosIOFoundInConfig: ARRAY[1..iMAX_SERCOS_IO] OF BOOL;
	udiNoOfElements: UDINT;
	udiNoOfElements2: UDINT;
	uiBufferPos: UINT;
	fbFileWriteAsync: SysFileWriteAsync;
END_VAR
VAR_INPUT
	/// start FB
	IN_bExecute: BOOL;
	/// Check if found axes = configured axes.
	IN_bCheckAxesConfig: BOOL := FALSE;
	/// Check if found sercos IO = configured sercos IO.
	IN_bCheckSercosIOConfig: BOOL := FALSE;
	/// Check if found module on sercos IO = configured module on sercos IO.
	IN_bCheckSercosIOModuleConfig: BOOL := FALSE;
	/// Check if found Inline IO = configured Inline IO.
	IN_bCheckInlineIOConfig: BOOL := FALSE;
	/// Write Sercos Address to IO
	IN_bWriteSercosIOAddress: BOOL := FALSE;
	/// Write Axes configuration to A-0-0024 
	IN_bConfigAxes: BOOL := FALSE;
	/// Write sercos IO configuration to C-0-0478 and UserDefs.cfg
	IN_bConfigSercosIO: BOOL := FALSE;
	/// Write Inline IO configuration to UserDefs.cfg	
	IN_bConfigInlineIO: BOOL := FALSE;
	/// Write Profibus IO configuration to UserDefs.cfg
	IN_bConfigProfibusIO: BOOL := FALSE;
	/// Write Profinet IO configuration to UserDefs.cfg
	IN_bConfigPNIO: BOOL := FALSE;
	/// Reboot automatically if necessary
	IN_bRebootAuto: BOOL := FALSE;
	/// Command Configuration of Devices
	IN_stDeviceCmdConfig: REFERENCE TO ST_DeviceCmdConfig;
	/// actual Configuration of Devices
	IN_stDeviceActConfig: REFERENCE TO ST_DeviceActConfig;
	IN_stDeviceConfigError: REFERENCE TO ST_DeviceConfigError;
END_VAR


IF IN_bExecute AND NOT bExecuteOld THEN
	bExecuteOld := TRUE;
	OUT_bActive := TRUE;
	OUT_bDone := FALSE;
	OUT_bError := FALSE;	
	sDiagMessageInt := '';
	OUT_sDiagMessage :='';
	
	// Referenzen aktualisieren
	refastAxesCmdConfig REF= IN_stDeviceCmdConfig.astAxes;
	refastInlineIOCmdConfig REF= IN_stDeviceCmdConfig.astInlineIO;
	refastSercosIOCmdConfig	REF= IN_stDeviceCmdConfig.astSercosIO;
	refastPNIOCmdConfig REF= IN_stDeviceCmdConfig.astPN_IO;
	
	refastAxesActConfig REF= IN_stDeviceActConfig.astAxes;
//	S20IOActConfig REF= DeviceActConfig.S20_IO;
	refastSercosIOActConfig	REF= IN_stDeviceActConfig.astSercosIO;
//	PNIOActConfig REF= DeviceActConfig.PN_IO;
	
	refastAxesConfigError REF= IN_stDeviceConfigError.astAxes;
	refastSercosIOConfigError REF= IN_stDeviceConfigError.astSercosIO;
//	SercosIOCmdConfigError REF= DeviceConfigError.sercos_IO_CmdConfig;
	refastFoundDrivesError REF=	IN_stDeviceConfigError.astFoundDrives;
	refastInlineIOConfigError REF= IN_stDeviceConfigError.astInlineIO;
	
	iState := 10;
ELSIF NOT IN_bExecute AND (OUT_bDone OR OUT_bError) THEN
	bExecuteOld := FALSE;
	OUT_bReboot := FALSE;
	OUT_bActive := FALSE;
	OUT_bDone := FALSE;
	OUT_bError := FALSE;	
	iState := 0;
END_IF


(* Now in Execute-Method
IF iState >= 10 AND iState < 100 THEN 
	THIS^.M_0ReadActConfig();
ELSIF iState >= 1000 AND iState < 1100 THEN
//	act11_DownloadDriveFirmware();				// Execute this Action in a different Task
 	iState := 100; 
ELSIF iState >= 100 AND iState < 200 THEN
	THIS^.M_1ConfigAxes();
ELSIF iState >= 200 AND iState < 300 THEN
	THIS^.M_2ConfigSercosIO();
ELSIF iState >= 300 AND iState < 400 THEN
	THIS^.M_3ConfigInlineIO();	
ELSIF iState >= 400 AND iState < 500 THEN
	THIS^.M_4ConfigProfibsIO();
ELSIF iState >= 500 AND iState < 600 THEN
	iState := 800;
ELSIF iState >= 800 AND iState < 900 THEN
	THIS^.M_8WriteConfig();
ELSIF iState >= 900 AND iState < 1000 THEN
	THIS^.M_9ErrorDone();
END_IF	
*)

METHOD PRIVATE _M_WriteLnString : DINT
VAR_INPUT
	/// file handle 
	dwHandle: DWORD;
	/// argument for format string 
	sArg: STRING(255);
END_VAR
VAR
	/// format string 
	sFormat: STRING(20) := '%s$R$N';
END_VAR
_M_WriteLnString := SysFileStreamFPrintf_String(dwHandle, sFormat, ADR(sArg));
END_METHOD

METHOD M_0ReadActConfig : BOOL


CASE iState OF
	
(* ################################################################################ *)	
	// Idle
(* ################################################################################ *)	
	0:
		OUT_bDone := FALSE;
		OUT_bError := FALSE;
		bErrorTemp := FALSE;
		OUT_bActive := FALSE;

(* ################################################################################ *)	
	// Reset FB
(* ################################################################################ *)	

	10://Start
	fbCommand (Execute	:= FALSE,
				Axis 	:= NoAxis);
	fbReadListParameter(Execute	:= FALSE,
				Axis 	:= NoAxis); 
	WriteC578(Execute	:= FALSE,
				Axis	:= NoAxis);
	fbWriteC506(Execute:=FALSE, 
				Axis:= 	NoAxis);				

	// delete old structure	
	FOR i := 1 TO iMAX_AXES_NUMBER DO
		// copy emty structure to initialize everything with default value
		refastAxesActConfig[i]:=	stDummyAxesActConfig;		
	END_FOR	
	FOR i := 1 TO iMAX_INLINE_IO DO
		M_DelStructure(IN_pbToElement:=ADR(refastInlineIOActConfig[i]) , IN_uiNoOfByte:=SIZEOF(refastInlineIOActConfig[i]) );
		M_DelStructure(IN_pbToElement:=ADR(InlineIOCfg[i]) , IN_uiNoOfByte:=SIZEOF(InlineIOCfg[i]) );		
	END_FOR	
	FOR i := 1 TO iMAX_SERCOS_IO DO
		M_DelStructure(IN_pbToElement:=ADR(refastSercosIOActConfig[i]) , IN_uiNoOfByte:=SIZEOF(refastSercosIOActConfig[i]) );
	END_FOR	
(*FOR i := 1 TO MAX_PROFIBUS_MASTER DO
		FOR j := 1 TO MAX_PROFIBUS_SLAVE DO
			M_DelStructure(PtrToElement:=ADR(ProfibusIOActConfig[i,j]) , NoOfByte:=SIZEOF(ProfibusIOActConfig[i,j]) );
		END_FOR	
	END_FOR	
*)	
	M_DelStructure(ADR(asAxisString), SIZEOF(asAxisString));
	M_DelStructure(ADR(aiC484), SIZEOF(aiC484));
	M_DelStructure(ADR(aiC510), SIZEOF(aiC510));
	M_DelStructure(ADR(apiPointerToC510), SIZEOF(apiPointerToC510));
	M_DelStructure(ADR(refastAxesConfigError), SIZEOF(refastAxesConfigError));
	M_DelStructure(ADR(refastFoundDrivesError), SIZEOF(refastFoundDrivesError));
	M_DelStructure(ADR(sRingString), SIZEOF(sRingString));
	M_DelStructure(ADR(sRingString2), SIZEOF(sRingString2));
	M_DelStructure(ADR(apsElements), SIZEOF(apsElements));
	M_DelStructure(ADR(apsElements2), SIZEOF(apsElements2));
	M_DelStructure(ADR(refastSercosIOActConfigC578), SIZEOF(refastSercosIOActConfigC578));
	
	fbINLNModuleConfigList(
		Execute:= FALSE, 
		SizeOfModuleConfig:=  SIZEOF(InlineIOCfg), 
		ModuleConfigAdr:= ADR(InlineIOCfg), 
		Done=> , 
		Active=> , 
		Error=> , 
		ErrorID=> , 
		ErrorIdent=> , 
		NoOfModuleConfig=> udiNoOfModuleConfig  );
	
	udiNoOfModuleConfig := 0;	
	
	iActNoOfDrives := 0;

	iState 	:= 15;
		
(* ################################################################################ *)	
	// Change sercos F8 Error reaction to F5
(* ################################################################################ *)	
//12:	
//	IF UpdateFirmware THEN
//		IF (NOT SercosErrorReaction.F2_Error AND NOT SercosErrorReaction.F5_Error AND NOT SercosErrorReaction.F8_Error)
//			OR SercosErrorReaction.F8_Error THEN
//			dwC506.0 := TRUE;		// for FWA Update change Error Reaction to F5
//			dwC506.1 := FALSE;
//		ELSIF SercosErrorReaction.F5_Error THEN
//			dwC506.0 := TRUE;
//			dwC506.1 := FALSE;
//		ELSIF SercosErrorReaction.F2_Error THEN  
//			dwC506.0 := FALSE;
//			dwC506.1 := TRUE;	
//		END_IF
//		
//		dwC506.7 := SercosErrorReaction.NoRedundancyWarning;
//		dwC506.8 := SercosErrorReaction.AutoRingRecovery; 
//		
//		fbWriteC506(
//			Execute:=TRUE , 
//			Done=> , 
//			Active=> , 
//			Error=> , 
//			ErrorID=> , 
//			ErrorIdent=> , 
//			ParameterNumber:= FP_C_0_0506, 
//			Value:= 	dwC506, 
//			Axis:= 	NoAxis);
//	END_IF
//	
//	IF fbWriteC506.Done OR NOT UpdateFirmware THEN
//		fbWriteC506(Execute:=FALSE, 
//				Axis:= 	NoAxis);	
//		iState 	:= 15;		
//	ELSIF fbWriteC506.Error then
//		ErrorID 	:= fbWriteC506.ErrorID;
//		ErrorIdent 	:= fbWriteC506.ErrorIdent;
//		fbWriteC506(Execute:=FALSE, 
//					Axis:= 	NoAxis);	
//		iState 		:= 998;
//	END_IF	
	
(* ################################################################################ *)	
	// Read actual configuration C-0-0578
(* ################################################################################ *)			
	15:
		fbReadListParameter(
			Execute			:= TRUE, 
			ParameterNumber	:= GVL_C_Param_ID.FP_C_0_0578, 
			NoOfBytes		:= SIZEOF(sRingString), 
			ValueAdr		:= ADR(sRingString), 
			Axis			:= NoAxis);
			
			IF fbReadListParameter.Done THEN
				fbReadListParameter(Execute	:= FALSE,
									Axis	:= NoAxis);
				iState 	:= 20;
				
				// split String																//Workaround Defdb00192639, -1 if string is empty					
				udiNoOfElements := IL_StrSplit(ADR(sRingString),',',0,FALSE,ADR(apsElements),TO_UDINT(SIZEOF(apsElements) - TO_INT(NOT TO_BOOL(LEN(sRingString)))) );
				//					IL_StrSplit(ADR(sRingString),',',0,FALSE,ADR(arElements),TO_UDINT(SIZEOF(arElements) - TO_INT(NOT TO_BOOL(LEN(sRingString)))) ); 
				{warning 'JS: strSplit'}
				//strSplit(ADR(sRingString),CHAR_COMMA,0,FALSE,ADR(arElements));
			ELSIF fbReadListParameter.Error THEN
				OUT_ErrorID 	:= fbReadListParameter.ErrorID;
				OUT_ErrorIdent 	:= fbReadListParameter.ErrorIdent;
				fbReadListParameter(Execute	:= FALSE,
									Axis	:= NoAxis);
				iState 		:= 998;
			END_IF
				
(* ################################################################################ *)	
	// copy IO configuration C-0-0578 into structure
(* ################################################################################ *)			
	20:	
 		i := 0;
		j := 1;
		k := 1;
		
		//copy string into structure
		FOR i := 0 TO (TO_INT(udiNoOfElements/iMAX_NUM_ELEMENTS_C578)-1) DO 
		//REPEAT
			//Delete 'A' at beginning of String
			IF (apsElements[iMAX_NUM_ELEMENTS_C578*i+1]^ <> '') THEN
				psString := apsElements[iMAX_NUM_ELEMENTS_C578*i+1]+1;
			ELSE
				psString := apsElements[iMAX_NUM_ELEMENTS_C578*i+1];
			END_IF
			
			iSercosAddressTemp :=  STRING_TO_INT(psString^);
			psRingString2 := apsElements[iMAX_NUM_ELEMENTS_C578*i+2];
	//		sRingString2 := ptrRingString2^; 
	//		strSplit(ADR(sRingString2),CHAR_MINUS,0,FALSE,ADR(arElements2));
				
			// sercos IO
			IF 	M_TypeCodeIsRexrothIO(sTypeCode:=LEFT (apsElements[iMAX_NUM_ELEMENTS_C578*i+3]^,13) ) THEN
				refastSercosIOActConfigC578[j].bAvailable := TRUE;
				refastSercosIOActConfigC578[j].iSercosAddress := iSercosAddressTemp;
			
				refastSercosIOActConfigC578[j].sTypeCode 	:= RIGHT (apsElements[iMAX_NUM_ELEMENTS_C578*i+3]^,10);
				j := j + 1;
			END_IF
	
	//	UNTIL(arElements[MAX_NUM_ELEMENTS_C578*i+1]^ = '' OR i >= MAX_SERCOS_DEVICES )
	//	END_REPEAT
		END_FOR
		
		M_DelStructure(ADR(sRingString), SIZEOF(sRingString));
		M_DelStructure(ADR(sRingString2), SIZEOF(sRingString2));
		M_DelStructure(ADR(apsElements), SIZEOF(apsElements));
		M_DelStructure(ADR(apsElements2), SIZEOF(apsElements2));
		
		iState 		:= 25;
	
(* ################################################################################ *)	
	// Refresh FP_C_0_0479
(* ################################################################################ *)	
	25:
	fbCommand(	Execute			:= TRUE, 
				ParameterNumber	:= GVL_C_Param_ID.FP_C_0_1009, 
				Axis			:= NoAxis);

	IF fbCommand.Done THEN
		fbCommand(	Execute	:= FALSE,
					Axis	:= NoAxis);
		iState	:= 30;
	ELSIF fbCommand.Error THEN
		OUT_ErrorID		:= fbCommand.ErrorID;
		OUT_ErrorIdent	:= fbCommand.ErrorIdent;
		fbCommand(	Execute:= FALSE,
					Axis:= NoAxis);
		iState 		:= 998;
	END_IF	
	
(* ################################################################################ *)	
	//read connected sercos devices
(* ################################################################################ *)	
	30:
		fbReadListParameter(
			Execute			:= TRUE, 
			ParameterNumber	:= GVL_C_Param_ID.FP_C_0_0479, 
			NoOfBytes		:= SIZEOF (sRingString), 
			ValueAdr		:= ADR(sRingString), 
			Axis			:= NoAxis);
			
			IF fbReadListParameter.Done THEN
				fbReadListParameter(Execute	:= FALSE,
									Axis	:= NoAxis);
				iState 	:= 35;
			ELSIF fbReadListParameter.Error THEN
				OUT_ErrorID 	:= fbReadListParameter.ErrorID;
				OUT_ErrorIdent 	:= fbReadListParameter.ErrorIdent;
				fbReadListParameter(Execute	:= FALSE,
									Axis	:= NoAxis);
				iState 		:= 998;
			END_IF

		
(* ################################################################################ *)	
	//read configured drives
(* ################################################################################ *)				
	35: 
		fbReadListParameter(
			Execute			:= TRUE, 
			ParameterNumber	:= GVL_C_Param_ID.FP_C_0_0484, 
			NoOfBytes		:= SIZEOF(aiC484), 
			ValueAdr		:= ADR(aiC484), 
			Axis			:= NoAxis);
			
			IF fbReadListParameter.Done THEN
				fbReadListParameter(Execute	:= FALSE,
									Axis	:= NoAxis);
				iState 	:= 38;
			ELSIF fbReadListParameter.Error THEN
				OUT_ErrorID 	:= fbReadListParameter.ErrorID;
				OUT_ErrorIdent 	:= fbReadListParameter.ErrorIdent;
				fbReadListParameter(Execute	:= FALSE,
									Axis	:= NoAxis);
				iState 		:= 998;
			END_IF
		
(* ################################################################################ *)	
	//read Sercos address configuration
(* ################################################################################ *)					
	38:
		fbReadListParameter(
			Execute			:= TRUE, 
			ParameterNumber	:= GVL_C_Param_ID.FP_C_0_0510, 
			NoOfBytes		:= SIZEOF(aiC510), 
			ValueAdr		:= ADR(aiC510), 
			Axis			:= NoAxis,
			NoOfRecBytes	=> uiLengthArC510 );
		
		IF fbReadListParameter.Done THEN
			fbReadListParameter(Execute	:= FALSE,
								Axis	:= NoAxis);
			iState 	:= 40;
		ELSIF fbReadListParameter.Error THEN
			OUT_ErrorID 	:= fbReadListParameter.ErrorID;
			OUT_ErrorIdent 	:= fbReadListParameter.ErrorIdent;
			fbReadListParameter(Execute	:= FALSE,
								Axis	:= NoAxis);
			iState 		:= 998;
		END_IF

			
(* ################################################################################ *)	
	//split and copy the string into a structure
(* ################################################################################ *)					
	40:	
 		i := 0;
		j := 1;
		k := 1;
		
		// split String																//Workaround Defdb00192639, -1 if string is empty					
		udiNoOfElements := IL_StrSplit(ADR(sRingString),',',0,FALSE,ADR(apsElements),TO_UDINT(SIZEOF(apsElements) - TO_INT(NOT TO_BOOL(LEN(sRingString)))) );
				
		
		//split
		// IL_StrSplit(ADR(sRingString),',',0,FALSE,ADR(arElements),TO_UDINT(SIZEOF(arElements) - TO_INT(NOT TO_BOOL(LEN(sRingString)))) ); 
		{warning 'JS: strSplit'}
		//strSplit(ADR(sRingString),CHAR_COMMA,0,FALSE,ADR(arElements));
		//copy string into structure
		//REPEAT
		FOR i := 0 TO (TO_INT(udiNoOfElements/iMAX_NUM_ELEMENTS_C479)-1) DO 
			//Delete 'A' at beginnin of String
			IF (apsElements[iMAX_NUM_ELEMENTS_C479*i+1]^ <> '') THEN
				psString := apsElements[iMAX_NUM_ELEMENTS_C479*i+1]+1;
			ELSE
				psString := apsElements[iMAX_NUM_ELEMENTS_C479*i+1];
			END_IF
			
			iSercosAddressTemp :=  STRING_TO_INT(psString^);
			psRingString2 := apsElements[iMAX_NUM_ELEMENTS_C479*i+2];
			sRingString2 := psRingString2^;

			// split String																						//Workaround Defdb00192639, -1 if string is empty	
			udiNoOfElements2 := IL_StrSplit(ADR(sRingString2),'-',0,FALSE,ADR(apsElements2),TO_UDINT(SIZEOF(apsElements2) - TO_INT(NOT TO_BOOL(LEN(sRingString2)))) );
			//IL_StrSplit(ADR(sRingString2),'-',0,FALSE,ADR(arElements2),TO_UDINT(SIZEOF(arElements2) - TO_INT(NOT TO_BOOL(LEN(sRingString2)))) ); 
			{warning 'JS: strSplit'}
			//strSplit(ADR(sRingString2),CHAR_MINUS,0,FALSE,ADR(arElements2));
			

			// check length
			IF udiNoOfElements > 7 THEN 	
				// sercos IO
				IF 	M_TypeCodeIsRexrothIO(sTypeCode:=LEFT (apsElements[iMAX_NUM_ELEMENTS_C479*i+7]^,13) ) THEN
					refastSercosIOActConfig[j].bAvailable := TRUE;
					refastSercosIOActConfig[j].iSercosAddress := iSercosAddressTemp;
				
					refastSercosIOActConfig[j].sTypeCode 		:= RIGHT(apsElements[iMAX_NUM_ELEMENTS_C479*i+7]^,10);
					
				// Where are I/O addresses in C-0-0510
					apiPointerToC510[j] := ADR (aiC510[i+1]);	
					j := j +1;			
				
				// Axis
				ELSIF LEFT (apsElements[iMAX_NUM_ELEMENTS_C479*i+2]^,4) = 'FFWA' THEN
					refastAxesActConfig[k].bRealAxis 			:= TRUE;
					refastAxesActConfig[k].bAvailable 			:= TRUE;		
					refastAxesActConfig[k].iSercosAddress := iSercosAddressTemp;	
					
					// copy Firmware to structure (6 characters)
					sTemp := '-';
					IL_CONCAT(ADR(refastAxesActConfig[k].sFirmware), apsElements2[3], ADR(refastAxesActConfig[k].sFirmware), 8);
					IL_CONCAT(ADR(refastAxesActConfig[k].sFirmware), ADR(sTemp), ADR(refastAxesActConfig[k].sFirmware), 8);
					sTemp := '';
	
